# B&R Automation Studio project PT_KB_V01 (part 2)

#### Types.typ - Exported data types
```iecst
(* ============================================================================ *)
(* BR_LIB - CENTRALNI PREGLED SVIH DATA TYPE DEKLARACIJA                       *)
(* Sadrzi TYPE deklaracije iz FB-ova koje smo standardizovali.                  *)
(* Namena: referenca, copy/paste i priprema za eventualno centralno tipiziranje.*)
(* ============================================================================ *)

TYPE
	(* ======================================================================== *)
	(* FB_AI_01_DI_01                                                         *)
	(* ======================================================================== *)
	typInAI01_DI01 : STRUCT (* Ulazna struktura FB_AI_01_DI_01. *)
		Enable : BOOL; (* Globalni enable FB-a *)
		RawValue : INT; (* Raw vrednost sa AI kanala *)
		ManualValue : REAL; (* Rucno zadana skalirana vrednost *)
		EnableManual : BOOL; (* TRUE = koristi ManualValue umesto RawValue *)
		ResetAlarm : BOOL; (* Reset latched alarma *)
		ManualAlarm : BOOL; (* Spoljasnji/manual alarm signal *)
		UnderRange : BOOL; (* Sistemski signal: ulaz ispod opsega *)
		OverRange : BOOL; (* Sistemski signal: ulaz iznad opsega *)
		TransmitterStatus : BOOL; (* TRUE = transmiter ispravan; FALSE = fault sa transmitera *)
	END_STRUCT;

	typParAI01_DI01 : STRUCT (* Parametarska struktura FB_AI_01_DI_01. *)
		RawMin : INT; (* Donja granica raw opsega *)
		RawMax : INT; (* Gornja granica raw opsega *)
		ScaledMin : REAL; (* Donja granica skaliranog opsega *)
		ScaledMax : REAL; (* Gornja granica skaliranog opsega *)
		EnableStatusCheck : BOOL; (* TRUE = koristi TransmitterStatus u logici; FALSE = ignorise statusni DI signal *)
		UnitOfMeasure : STRING[80]; (* Jedinica mere za izlaznu vrednost *)
	END_STRUCT;

	typOutAI01_DI01 : STRUCT (* Izlazna struktura FB_AI_01_DI_01. *)
		ScaledValue : REAL; (* Skalirana inzenjerska vrednost *)
		Status : BOOL; (* TRUE = FB je omogucen, bez Stop-a, blokirajuceg fault-a i re-enable zahteva. *)
		State : USINT; (* Numericki kod stanja *)
		State_comment : STRING[80]; (* Trenutni opis stanja *)
		UnitOfMeasureOut : STRING[80]; (* Prosledjena jedinica mere *)
		TransmitterStatusIn : BOOL; (* Kopija ulaznog statusnog signala transmitera za HMI/SCADA *)
		FaultLatched : BOOL; (* Memorisan fault do validnog reset-a. *)
		FaultCondition : BOOL; (* Trenutni fault uslov u ovom scan-u. *)
		ResetAllowed : BOOL; (* TRUE kada fault moze biti resetovan bez ponovnog latche-ovanja. *)
		ConfigValid : BOOL; (* TRUE kada su opsezi validno konfigurirani. *)
		ConfigFaultText : STRING[80]; (* Opis prve nevalidne konfiguracije parametara. *)
		FaultCode : USINT; (* Kod memorisanog fault uzroka. *)
		FaultText : STRING[80]; (* Tekst memorisanog fault uzroka. *)
		Diag : STRING[80]; (* Kratak operativni tekst za HMI nadzor. *)
	END_STRUCT;

	typIntAI01_DI01 : STRUCT (* Interna radna struktura FB_AI_01_DI_01. *)
		FaultLatched : BOOL; (* Memorisan alarm dok se ne resetuje *)
		FaultCondition : BOOL; (* Trenutni fault uslov u ovom scan-u *)
		ActiveFaultCode : USINT; (* Trenutni aktivni fault kod u ovom scan-u. *)
		ScaleSpanRaw : REAL; (* Raspon raw opsega *)
		ScaleSpanScaled : REAL; (* Raspon skaliranog opsega *)
		ManualValueLimited : REAL; (* Ogranicena manual vrednost na parametarski opseg *)
		ResetRequest : BOOL; (* Interna kopija reset komande *)
		ResetAllowed : BOOL; (* Interna dozvola reset-a latched fault-a. *)
		ConfigValid : BOOL; (* FALSE kada opsezi nisu validno konfigurisani. *)
		ConfigFaultText : STRING[80]; (* Tekst prve nevalidne konfiguracije. *)
		FaultCode : USINT; (* Memorisani fault kod. *)
		FaultText : STRING[80]; (* Tekst memorisanog fault uzroka. *)
		Diag : STRING[80]; (* Interna dijagnostika trenutnog rezima i fault stanja. *)
	END_STRUCT;

	typConstAI01_DI01 : STRUCT (* Struktura konstanti i state tekstova FB_AI_01_DI_01. *)
		ST_DISABLED : USINT := 0; (* Blok onemogucen (Enable=FALSE). *)
		ST_ACTIVE : USINT := 1; (* Normalan rad bez alarma. *)
		ST_UNDERRANGE : USINT := 2; (* Raw vrednost ispod RawMin granice. *)
		ST_OVERRANGE : USINT := 3; (* Raw vrednost iznad RawMax granice. *)
		ST_FAULT : USINT := 4; (* Latched fault stanje u automatskom radu. *)
		ST_MANUAL : USINT := 5; (* Aktivno manuelno zadavanje bez fault-a. *)
		ST_MANUAL_FAULT : USINT := 6; (* Manuelni rad uz aktivan latched fault. *)
		ST_TRANSMITTER_STATUS_0 : USINT := 7; (* Statusni DI transmitera je FALSE. *)
		FLT_NONE : USINT := 0; (* Nema aktivnog fault uzroka. *)
		FLT_MANUAL_ALARM : USINT := 1; (* ManualAlarm ulaz je aktivan. *)
		FLT_UNDERRANGE : USINT := 2; (* UnderRange signal je aktivan. *)
		FLT_OVERRANGE : USINT := 3; (* OverRange signal je aktivan. *)
		FLT_CONFIG_INVALID : USINT := 4; (* Parametri opsega su nevalidni. *)
		CMT_DISABLED : STRING[80] := 'Stanje 0: transmiter neaktivan (Enable=FALSE), izlaz je na 0.0.'; (* Tekstualni opis stanja ST_DISABLED. *)
		CMT_ACTIVE : STRING[80] := 'Stanje 1: normalan rad, ulaz je u dozvoljenom opsegu, bez alarma.'; (* Tekstualni opis stanja ST_ACTIVE. *)
		CMT_UNDERRANGE : STRING[80] := 'Stanje 2: ulazna raw vrednost je ispod definisanog minimuma (RawMin).'; (* Tekstualni opis stanja ST_UNDERRANGE. *)
		CMT_OVERRANGE : STRING[80] := 'Stanje 3: ulazna raw vrednost je iznad definisanog maksimuma (RawMax).'; (* Tekstualni opis stanja ST_OVERRANGE. *)
		CMT_FAULT : STRING[80] := 'Stanje 4: prisutan je alarm (latched), potreban je ResetAlarm za potvrdu.'; (* Tekstualni opis stanja ST_FAULT. *)
		CMT_MANUAL : STRING[80] := 'Stanje 5: aktivan rucni rezim, ScaledValue dolazi iz ManualValue.'; (* Tekstualni opis stanja ST_MANUAL. *)
		CMT_MANUAL_FAULT : STRING[80] := 'Stanje 6: aktivan rucni rezim i istovremeno prisutan latched alarm.'; (* Tekstualni opis stanja ST_MANUAL_FAULT. *)
		CMT_TRANSMITTER_STATUS_0 : STRING[80] := 'Stanje 7: statusni DI signal transmitera je 0 (EnableStatusCheck=TRUE).'; (* Tekstualni opis stanja ST_TRANSMITTER_STATUS_0. *)
	END_STRUCT;

	typAI01_DI01 : STRUCT (* Agregatna struktura svih sekcija za FB_AI_01_DI_01. *)
		Input : typInAI01_DI01; (* Ulazni signali i komande bloka. *)
		Param : typParAI01_DI01; (* Parametri skaliranja i ponasanja. *)
		Output : typOutAI01_DI01; (* Izlazi, status i state informacije. *)
		Internal : typIntAI01_DI01; (* Interna radna memorija. *)
		Constant : typConstAI01_DI01; (* Konstante state kodova i tekstova. *)
	END_STRUCT;

	(* ======================================================================== *)
	(* FB_AI_01_DI_01_DO_02                                                    *)
	(* ======================================================================== *)
	typInAI01_DI01_DO02 : STRUCT (* Ulazna struktura FB_AI_01_DI_01_DO_02. *)
		Enable : BOOL; (* Globalni enable FB-a *)
		RawValue : INT; (* Raw vrednost sa AI kanala *)
		ManualValue : REAL; (* Rucno zadana skalirana vrednost *)
		EnableManual : BOOL; (* TRUE = koristi ManualValue umesto RawValue *)
		ResetAlarm : BOOL; (* Reset latched alarma *)
		ManualAlarm : BOOL; (* Spoljasnji/manual alarm signal *)
		UnderRange : BOOL; (* Sistemski signal: ulaz ispod opsega *)
		OverRange : BOOL; (* Sistemski signal: ulaz iznad opsega *)
		TransmitterStatus : BOOL; (* TRUE = transmiter ispravan; FALSE = fault sa transmitera *)
		RangeSelect : USINT; (* Izbor opsega 1..4 *)
		RangeSettleTime : TIME; (* Vreme stabilizacije nakon promene opsega *)
	END_STRUCT;

	typParAI01_DI01_DO02 : STRUCT (* Parametarska struktura FB_AI_01_DI_01_DO_02. *)
		RawMin : INT; (* Donja granica raw opsega *)
		RawMax : INT; (* Gornja granica raw opsega *)
		ScaledMin_R1 : REAL; (* Donja granica skaliranog opsega R1 *)
		ScaledMax_R1 : REAL; (* Gornja granica skaliranog opsega R1 *)
		ScaledMin_R2 : REAL; (* Donja granica skaliranog opsega R2 *)
		ScaledMax_R2 : REAL; (* Gornja granica skaliranog opsega R2 *)
		ScaledMin_R3 : REAL; (* Donja granica skaliranog opsega R3 *)
		ScaledMax_R3 : REAL; (* Gornja granica skaliranog opsega R3 *)
		ScaledMin_R4 : REAL; (* Donja granica skaliranog opsega R4 *)
		ScaledMax_R4 : REAL; (* Gornja granica skaliranog opsega R4 *)
		UnitOfMeasure : STRING[80]; (* Jedinica mere za izlaznu vrednost *)
	END_STRUCT;

	typOutAI01_DI01_DO02 : STRUCT (* Izlazna struktura FB_AI_01_DI_01_DO_02. *)
		ScaledValue : REAL; (* Skalirana inzenjerska vrednost *)
		Status : BOOL; (* TRUE = bez alarma i Enable=TRUE *)
		State : USINT; (* Numericki kod stanja *)
		State_comment : STRING[80]; (* Trenutni opis stanja *)
		UnitOfMeasureOut : STRING[80]; (* Prosledjena jedinica mere *)
		TransmitterStatusIn : BOOL; (* Kopija ulaznog statusnog signala transmitera za HMI/SCADA *)
		ActiveRange : USINT; (* Trenutno aktivan opseg 1..4 *)
		RangeComment : STRING[40]; (* Opis aktivnog opsega *)
		RangeBit0_out : BOOL; (* DO bit 0 za izbor opsega *)
		RangeBit1_out : BOOL; (* DO bit 1 za izbor opsega *)
		RangeChanging : BOOL; (* TRUE tokom stabilizacije promene opsega *)
		FaultProcessOut : BOOL; (* TRUE kada je aktivan procesni fault *)
		FaultConfigOut : BOOL; (* TRUE kada je aktivan konfiguracioni fault *)
	END_STRUCT;

	typIntAI01_DI01_DO02 : STRUCT (* Interna radna struktura FB_AI_01_DI_01_DO_02. *)
		FaultLatched : BOOL; (* Memorisan alarm dok se ne resetuje *)
		FaultCondition : BOOL; (* Trenutni fault uslov u ovom scan-u *)
		FaultProcess : BOOL; (* Procesni fault: DI status i under/over-range *)
		FaultConfig : BOOL; (* Konfiguracioni fault: parametri i range izbor *)
		ScaleSpanRaw : REAL; (* Raspon raw opsega *)
		ScaleSpanScaled : REAL; (* Raspon aktivnog skaliranog opsega *)
		ManualValueLimited : REAL; (* Ogranicena manual vrednost na aktivan opseg *)
		ActiveScaledMin : REAL; (* Donja granica aktivnog opsega *)
		ActiveScaledMax : REAL; (* Gornja granica aktivnog opsega *)
		LastGoodScaledValue : REAL; (* Poslednja validna vrednost pre promene opsega *)
		PrevRangeSelect : USINT; (* Prethodno izabrani opseg *)
		RangeChangeMem : BOOL; (* Memorija promene opsega *)
		ResetRequest : BOOL; (* Interna kopija reset komande *)
		RangeSettleTimeEffective : TIME; (* Validiran PT za tajmer stabilizacije *)
		RangeSettleTimer : TON; (* Tajmer stabilizacije posle promene opsega *)
	END_STRUCT;

	typConstAI01_DI01_DO02 : STRUCT (* Struktura konstanti i state tekstova FB_AI_01_DI_01_DO_02. *)
		ST_DISABLED : USINT := 0; (* Blok onemogucen (Enable=FALSE). *)
		ST_ACTIVE : USINT := 1; (* Normalan rad bez alarma. *)
		ST_UNDERRANGE : USINT := 2; (* Raw vrednost ispod RawMin granice. *)
		ST_OVERRANGE : USINT := 3; (* Raw vrednost iznad RawMax granice. *)
		ST_FAULT : USINT := 4; (* Latched fault stanje u automatskom radu. *)
		ST_MANUAL : USINT := 5; (* Aktivno manuelno zadavanje bez fault-a. *)
		ST_MANUAL_FAULT : USINT := 6; (* Manuelni rad uz aktivan latched fault. *)
		ST_TRANSMITTER_STATUS_0 : USINT := 7; (* Statusni DI transmitera je FALSE. *)
		ST_RANGE_CHANGING : USINT := 8; (* U toku je stabilizacija nakon promene opsega. *)
		CMT_DISABLED : STRING[80] := 'Stanje 0: transmiter neaktivan (Enable=FALSE), izlaz je na 0.0.'; (* Tekstualni opis stanja ST_DISABLED. *)
		CMT_ACTIVE : STRING[80] := 'Stanje 1: normalan rad, ulaz je u dozvoljenom opsegu, bez alarma.'; (* Tekstualni opis stanja ST_ACTIVE. *)
		CMT_UNDERRANGE : STRING[80] := 'Stanje 2: ulazna raw vrednost je ispod definisanog minimuma (RawMin).'; (* Tekstualni opis stanja ST_UNDERRANGE. *)
		CMT_OVERRANGE : STRING[80] := 'Stanje 3: ulazna raw vrednost je iznad definisanog maksimuma (RawMax).'; (* Tekstualni opis stanja ST_OVERRANGE. *)
		CMT_FAULT : STRING[80] := 'Stanje 4: prisutan je alarm (latched), potreban je ResetAlarm za potvrdu.'; (* Tekstualni opis stanja ST_FAULT. *)
		CMT_MANUAL : STRING[80] := 'Stanje 5: aktivan rucni rezim, ScaledValue dolazi iz ManualValue.'; (* Tekstualni opis stanja ST_MANUAL. *)
		CMT_MANUAL_FAULT : STRING[80] := 'Stanje 6: aktivan rucni rezim i istovremeno prisutan latched alarm.'; (* Tekstualni opis stanja ST_MANUAL_FAULT. *)
		CMT_TRANSMITTER_STATUS_0 : STRING[80] := 'Stanje 7: statusni DI signal transmitera je 0; skaliranje ostaje aktivno.'; (* Tekstualni opis stanja ST_TRANSMITTER_STATUS_0. *)
		CMT_RANGE_CHANGING : STRING[80] := 'Stanje 8: promena opsega je u toku; ceka se stabilizacija opsega.'; (* Tekstualni opis stanja ST_RANGE_CHANGING. *)
	END_STRUCT;

	typAI01_DI01_DO02 : STRUCT (* Agregatna struktura svih sekcija za FB_AI_01_DI_01_DO_02. *)
		Input : typInAI01_DI01_DO02; (* Ulazi sa izborom opsega i komandama. *)
		Param : typParAI01_DI01_DO02; (* Parametri opsega i skaliranja. *)
		Output : typOutAI01_DI01_DO02; (* Izlazi, aktivan opseg i fault status. *)
		Internal : typIntAI01_DI01_DO02; (* Interne pomocne promenljive i tajmeri. *)
		Constant : typConstAI01_DI01_DO02; (* Konstante stanja i komentari stanja. *)
	END_STRUCT;

	(* ======================================================================== *)
	(* FB_DI                                                                    *)
	(* ======================================================================== *)
	typInDI : STRUCT (* Ulazna struktura FB_DI. *)
		Enable : BOOL; (* Globalni enable FB-a *)
		SensorIn : BOOL; (* Digitalni ulaz sa terena *)
		StatusIn : BOOL; (* Statusni signal uredjaja, opciono koristi logika *)
		EnableManual : BOOL; (* TRUE = koristi ManualValue umesto SignalIn *)
		ManualValue : BOOL; (* Rucno zadat DI signal *)
		ResetAlarm : BOOL; (* Reset latched alarma *)
		ManualAlarm : BOOL; (* Spoljasnji/manual alarm signal *)
	END_STRUCT;

	typParDI : STRUCT (* Parametarska struktura FB_DI. *)
		UseStatusInput : BOOL; (* TRUE = proverava StatusIn; FALSE = ignorise ga *)
		InvertSignal : BOOL; (* TRUE = invertuje ulaznu DI vrednost *)
		DelayOn : TIME; (* Vreme potvrde OFF->ON prelaza *)
		DelayOff : TIME; (* Vreme potvrde ON->OFF prelaza *)
		AlarmOnTrue : BOOL; (* Alarm aktivan kada je Value=TRUE *)
		AlarmOnFalse : BOOL; (* Alarm aktivan kada je Value=FALSE *)
		TextTrue : STRING[80]; (* Tekst za stanje Value=TRUE *)
		TextFalse : STRING[80]; (* Tekst za stanje Value=FALSE *)
		TextAlarm : STRING[80]; (* Tekst za alarm stanje *)
		TextFault : STRING[80]; (* Tekst za fault stanje *)
	END_STRUCT;

	typOutDI : STRUCT (* Izlazna struktura FB_DI. *)
		Value : BOOL; (* Finalna DI vrednost nakon manual/invert/delay obrade *)
		Status : BOOL; (* TRUE = Enable aktivan i nema latched fault-a. *)
		Alarm : BOOL; (* Procesni alarm prema AlarmOnTrue/AlarmOnFalse *)
		Error : BOOL; (* Fault latch izlaz *)
		ManualActive : BOOL; (* TRUE kada je manual rezim aktivan *)
		State : USINT; (* Numericki kod stanja *)
		State_comment : STRING[80]; (* Tekstualni opis stanja *)
		StatusSignalIn : BOOL; (* Kopija statusnog signala za HMI/SCADA *)
		FaultLatched : BOOL; (* Memorisan fault do validnog reset-a *)
		FaultCondition : BOOL; (* Trenutni fault uslov u ovom scan-u *)
		AlarmCondition : BOOL; (* Trenutni procesni alarm uslov *)
		ResetAllowed : BOOL; (* TRUE kada fault moze biti resetovan bez ponovnog latche-ovanja. *)
		ConfigValid : BOOL; (* TRUE kada su DelayOn i DelayOff parametri validni. *)
		ConfigFaultText : STRING[80]; (* Opis nevalidne konfiguracije parametara. *)
		FaultCode : USINT; (* Kod memorisanog fault uzroka. *)
		FaultText : STRING[80]; (* Tekst memorisanog fault uzroka. *)
		Diag : STRING[80]; (* Kratak operativni tekst za HMI nadzor. *)
	END_STRUCT;

	typIntDI : STRUCT (* Interna radna struktura FB_DI. *)
		SignalRaw : BOOL; (* Vrednost pre delay obrade *)
		SignalFiltered : BOOL; (* Vrednost nakon delay obrade *)
		FaultLatched : BOOL; (* Interni fault latch *)
		FaultCondition : BOOL; (* Interni fault uslov u scan-u *)
		AlarmCondition : BOOL; (* Interni procesni alarm uslov *)
		ConfigValid : BOOL; (* FALSE kada su DelayOn/DelayOff parametri nevalidni. *)
		ResetAllowed : BOOL; (* Interna dozvola reseta fault-a. *)
		FaultCode : USINT; (* Memorisani kod fault uzroka. *)
		FaultText : STRING[80]; (* Tekst memorisanog fault uzroka. *)
		Diag : STRING[80]; (* Interna dijagnostika trenutnog rezima i fault stanja. *)
		TonOn : TON; (* Delay ON tajmer *)
		TonOff : TON; (* Delay OFF tajmer *)
	END_STRUCT;

	typConstDI : STRUCT (* Struktura state konstanti FB_DI. *)
		ST_DISABLED : USINT := 0; (* Blok onemogucen. *)
		ST_AUTO_FALSE : USINT := 1; (* Auto rezim, izlazna vrednost FALSE. *)
		ST_AUTO_TRUE : USINT := 2; (* Auto rezim, izlazna vrednost TRUE. *)
		ST_AUTO_ALARM : USINT := 3; (* Auto rezim sa procesnim alarmom. *)
		ST_AUTO_FAULT : USINT := 4; (* Auto rezim sa fault stanjem. *)
		ST_MAN_FALSE : USINT := 5; (* Manual rezim, izlazna vrednost FALSE. *)
		ST_MAN_TRUE : USINT := 6; (* Manual rezim, izlazna vrednost TRUE. *)
		ST_MAN_ALARM : USINT := 7; (* Manual rezim sa procesnim alarmom. *)
		ST_MAN_FAULT : USINT := 8; (* Manual rezim sa fault stanjem. *)
		FLT_NONE : USINT := 0; (* Nema aktivnog fault uzroka. *)
		FLT_MANUAL_ALARM : USINT := 1; (* ManualAlarm ulaz je aktivan. *)
		FLT_STATUS_INPUT : USINT := 2; (* StatusIn fault kada je UseStatusInput aktivan. *)
		FLT_CONFIG_INVALID : USINT := 3; (* Delay parametri su nevalidni. *)
	END_STRUCT;

	typDI : STRUCT (* Agregatna struktura svih sekcija za FB_DI. *)
		Input : typInDI; (* Ulazni signali, manual i reset komande. *)
		Param : typParDI; (* Parametri obrade i tekstovi stanja. *)
		Output : typOutDI; (* Finalna DI vrednost, alarm/fault i stanje. *)
		Internal : typIntDI; (* Interna logika filtracije i latch-a. *)
		Constant : typConstDI; (* Konstante state kodova DI bloka. *)
	END_STRUCT;

	(* ======================================================================== *)
	(* FB_V_ON_OFF_FB                                                           *)
	(* ======================================================================== *)
	typInVOnOff : STRUCT (* Ulazna struktura FB_V_ON_OFF_FB. *)
		Enable : BOOL; (* Globalni enable FB-a *)
		Stop : BOOL; (* Operativni stop: odmah deaktivira kalem i zahteva novi Enable ciklus. *)
		EnableManual : BOOL; (* TRUE = komanda pozicije dolazi iz manual ulaza *)
		Open_Manual : BOOL; (* Manual zahtev: TRUE otvori, FALSE zatvori *)
		OpenFb : BOOL; (* Povratni signal otvorenog krajnjeg polozaja *)
		CloseFb : BOOL; (* Povratni signal zatvorenog krajnjeg polozaja *)
		ResetAlarm : BOOL; (* Reset memorisanog alarma, samo kada trenutni fault uslov nije aktivan *)
		ManualAlarm : BOOL; (* Spoljni/manual fault zahtev *)
		ForceCmd : BOOL; (* TRUE = komanda prolazi ka ventilu i u fault stanju; FALSE = komanda blokirana (bezbedan polozaj) *)
	END_STRUCT;

	typParVOnOff : STRUCT (* Parametarska struktura FB_V_ON_OFF_FB. *)
		DeEnergizedOpen : BOOL; (* TRUE = ventil je bez napajanja otvoren; FALSE = bez napajanja zatvoren. *)
		FbOpenExists : BOOL; (* TRUE ako fizicki postoji Open feedback signal *)
		FbCloseExists : BOOL; (* TRUE ako fizicki postoji Close feedback signal *)
		OpenMinTime : TIME; (* Minimalno dozvoljeno vreme otvaranja pre OpenFb potvrde *)
		OpenMaxTime : TIME; (* Maksimalno dozvoljeno vreme otvaranja do OpenFb potvrde *)
		CloseMinTime : TIME; (* Minimalno dozvoljeno vreme zatvaranja pre CloseFb potvrde *)
		CloseMaxTime : TIME; (* Maksimalno dozvoljeno vreme zatvaranja do CloseFb potvrde *)
		StableFbDelay : TIME; (* Delay za detekciju nestabilnog feedback-a u stabilnim stanjima *)
	END_STRUCT;

	typOutVOnOff : STRUCT (* Izlazna struktura FB_V_ON_OFF_FB. *)
		Cmd : BOOL; (* Komanda jednom kalemu; funkcija zavisi od DeEnergizedOpen. *)
		Opened : BOOL; (* FB trenutno koristi otvoren polozaj, fizicki potvrdjen ili vremenski pretpostavljen. *)
		Closed : BOOL; (* FB trenutno koristi zatvoren polozaj, fizicki potvrdjen ili vremenski pretpostavljen. *)
		PositionConfirmed : BOOL; (* Aktivni krajnji polozaj je potvrdjen odgovarajucim fizickim feedback-om. *)
		PositionAssumed : BOOL; (* Aktivni krajnji polozaj je vremenski pretpostavljen bez odgovarajuceg feedback-a. *)
		OpenAssumed : BOOL; (* Otvoren polozaj je vremenski pretpostavljen. *)
		CloseAssumed : BOOL; (* Zatvoren polozaj je vremenski pretpostavljen. *)
		Status : BOOL; (* TRUE = bez alarma i Enable=TRUE *)
		InTransition : BOOL; (* TRUE dok je ventil u stanjima ST_OPENING ili ST_CLOSING *)
		StopActive : BOOL; (* Kopija aktivnog operativnog Stop zahteva. *)
		WaitingReEnable : BOOL; (* FB ceka novi Enable FALSE->TRUE ciklus posle Stop-a ili fault reseta. *)
		ResetAllowed : BOOL; (* TRUE kada je dozvoljen reset latched alarma *)
		State : USINT; (* Kopija internog stanja za HMI *)
		State_comment : STRING[80]; (* Opis stanja za HMI *)
		Diag : STRING[40]; (* Kratka operativna dijagnostika za live nadzor *)
		FaultLatched : BOOL; (* Memorisan alarm, ostaje 1 do validnog reseta *)
		FaultCondition : BOOL; (* Trenutni fault uslov u ovom scan-u *)
		FaultInManual : BOOL; (* Alarm je nastao dok je bio aktivan manual mod *)
		FaultCode : USINT; (* Numericki kod alarma *)
		FaultText : STRING[80]; (* Tekst alarma za HMI *)
		ForceActive : BOOL; (* TRUE = blokirajuci fault je aktivan, a ForceCmd dozvoljava komandu. *)
		FeedbackAlarmCondition : BOOL; (* Trenutno nedostaje ocekivani stabilni feedback. *)
		FeedbackAlarmLatched : BOOL; (* Memorisan neblokirajuci alarm stabilnog feedback-a. *)
		FeedbackAlarmCode : USINT; (* Numericki kod neblokirajuceg feedback alarma. *)
		FeedbackAlarmText : STRING[80]; (* Tekst neblokirajuceg feedback alarma. *)
		ConfigFaultText : STRING[80]; (* Opis prve nevalidne konfiguracione vrednosti. *)
		LastOpenStartTime  : REAL; (* Vreme od Open komande do gubitka CloseFb [s]; 0.0 ako FbCloseExists=FALSE *)
		LastOpenTime       : REAL; (* Vreme od Open komande do OpenConfirm=TRUE [s]; 0.0 ako FbOpenExists=FALSE *)
		LastCloseStartTime : REAL; (* Vreme od ukidanja Open komande do gubitka OpenFb [s]; 0.0 ako FbOpenExists=FALSE *)
		LastCloseTime      : REAL; (* Vreme od ukidanja Open komande do CloseConfirm=TRUE [s]; 0.0 ako FbCloseExists=FALSE *)
	END_STRUCT;

	typIntVOnOff : STRUCT (* Interna radna struktura FB_V_ON_OFF_FB. *)
		DesiredOpen : BOOL; (* Zeljen polozaj ventila: TRUE = otvoren, FALSE = zatvoren *)
		CmdRequest : BOOL; (* Zahtev aktiviranja kalema nakon NC/NO konverzije. *)
		FaultLatched : BOOL; (* Memorisan alarm - ostaje aktivan dok se ne resetuje *)
		FaultCondition : BOOL; (* Trenutno aktivan uslov alarma u ovom ciklusu *)
		FaultInManual : BOOL; (* Pamti da li je alarm nastao u rucnom modu *)
		FaultCode : USINT; (* Interni broj greske *)
		FaultText : STRING[80]; (* Tekstualni opis greske za HMI *)
		OpenConfirm : BOOL; (* Potvrda da je ventil otvoren *)
		CloseConfirm : BOOL; (* Potvrda da je ventil zatvoren *)
		OpenAssumed : BOOL; (* Memorija vremenski pretpostavljenog otvorenog polozaja. *)
		CloseAssumed : BOOL; (* Memorija vremenski pretpostavljenog zatvorenog polozaja. *)
		FeedbackAlarmCondition : BOOL; (* Trenutni uslov neblokirajuceg feedback alarma. *)
		FeedbackAlarmLatched : BOOL; (* Memorisan neblokirajuci feedback alarm. *)
		FeedbackAlarmCode : USINT; (* Kod neblokirajuceg feedback alarma. *)
		ReEnableRequired : BOOL; (* Posle Stop-a ili fault reseta zahteva novi Enable rising edge. *)
		Step : USINT; (* Interno stanje state machine *)
		PrevEnable : BOOL; (* Pamti prethodno stanje Enable signala zbog detekcije rising edge *)
		OpeningStarted : BOOL; (* Tokom otvaranja: ventil je poceo da se otvara *)
		ClosingStarted : BOOL; (* Tokom zatvaranja: ventil je poceo da se zatvara *)
		StableClosedFbError : BOOL; (* U stabilno zatvorenom stanju postoji greska feedback-a *)
		StableOpenedFbError : BOOL; (* U stabilno otvorenom stanju postoji greska feedback-a *)
		OpenMinTimer : TON; (* Minimalno dozvoljeno vreme otvaranja *)
		OpenMaxTimer : TON; (* Maksimalno dozvoljeno vreme otvaranja *)
		CloseMinTimer : TON; (* Minimalno dozvoljeno vreme zatvaranja *)
		CloseMaxTimer : TON; (* Maksimalno dozvoljeno vreme zatvaranja *)
		OpenMeasureTimer : TON; (* Merenje realnog trajanja otvaranja *)
		CloseMeasureTimer : TON; (* Merenje realnog trajanja zatvaranja *)
		StableClosedFbTimer : TON; (* Delay za potvrdu greske feedback-a u zatvorenom stanju *)
		StableOpenedFbTimer : TON; (* Delay za potvrdu greske feedback-a u otvorenom stanju *)
		PrevCloseFb : BOOL; (* Prethodni scan CloseFb - za detekciju falling edge u ST_OPENING *)
		PrevOpenFb  : BOOL; (* Prethodni scan OpenFb  - za detekciju falling edge u ST_CLOSING *)
	END_STRUCT;

	typCfgVOnOff : STRUCT (* Konfiguraciona struktura state/fault kodova FB_V_ON_OFF_FB. *)
		OpenMinTime_Valid : TIME; (* Validirano minimalno vreme otvaranja. *)
		OpenMaxTime_Valid : TIME; (* Validirano maksimalno vreme otvaranja. *)
		CloseMinTime_Valid : TIME; (* Validirano minimalno vreme zatvaranja. *)
		CloseMaxTime_Valid : TIME; (* Validirano maksimalno vreme zatvaranja. *)
		StableFbDelay_Valid : TIME; (* Validiran delay nadzora stabilnog feedback-a. *)

		ST_DISABLED : USINT := 0; (* Blok onemogucen. *)
		ST_IDLE_CLOSED : USINT := 10; (* Stabilno stanje: ventil zatvoren. *)
		ST_IDLE_OPENED : USINT := 20; (* Stabilno stanje: ventil otvoren. *)
		ST_OPENING : USINT := 30; (* Tranzicija otvaranja u toku. *)
		ST_CLOSING : USINT := 40; (* Tranzicija zatvaranja u toku. *)
		ST_STOPPED : USINT := 50; (* Operativni Stop je aktivan. *)
		ST_WAIT_REENABLE : USINT := 60; (* Ceka se novi Enable FALSE->TRUE ciklus. *)
		ST_FAULT : USINT := 90; (* Fault stanje ventila. *)

		FLT_NONE : USINT := 0; (* Nema aktivnog fault-a. *)
		FLT_MANUAL_ALARM : USINT := 1; (* Manual alarm zahtev je aktivan. *)
		FLT_FB_CONFLICT : USINT := 2; (* Konflikt feedback-a (OpenFb i CloseFb). *)
		FLT_OPEN_TIMEOUT : USINT := 3; (* Otvaranje nije potvrdjeno u OpenMaxTime. *)
		FLT_OPEN_TOO_FAST : USINT := 4; (* Otvaranje potvrdeno pre OpenMinTime. *)
		FLT_CLOSE_TIMEOUT : USINT := 5; (* Zatvaranje nije potvrdjeno u CloseMaxTime. *)
		FLT_CLOSE_TOO_FAST : USINT := 6; (* Zatvaranje potvrdeno pre CloseMinTime. *)
		FLT_TIME_CONFIG_INVALID : USINT := 9; (* Nevalidna konfiguracija vremenskih parametara. *)

		FB_ALM_NONE : USINT := 0; (* Nema neblokirajuceg feedback alarma. *)
		FB_ALM_STABLE_OPEN_LOST : USINT := 1; (* Izgubljen OpenFb u stabilno otvorenom stanju. *)
		FB_ALM_STABLE_CLOSE_LOST : USINT := 2; (* Izgubljen CloseFb u stabilno zatvorenom stanju. *)
	END_STRUCT;

	(* ======================================================================== *)
	(* FB_V_EMV (elektromotorni ventil sa odvojenim OPEN/CLOSE komandama)       *)
	(* ======================================================================== *)
	typInVEmv : STRUCT (* Ulazna struktura FB_V_EMV. *)
		Enable : BOOL; (* Globalna dozvola rada FB-a. *)
		Stop : BOOL; (* Operativni stop: odmah gasi obe komande bez generisanja fault-a. *)
		EnableManual : BOOL; (* TRUE = koristi OpenManual umesto automatskog Open zahteva. *)
		OpenManual : BOOL; (* Manualni zahtev polozaja: TRUE = OPEN, FALSE = CLOSE. *)
		ForceCmd : BOOL; (* Dozvola kontrolisanog kretanja u suprotnom smeru iz fault-a. *)
		ResetAlarm : BOOL; (* Zahtev za reset latched fault-a kada su ispunjeni bezbedni uslovi. *)
		ManualAlarm : BOOL; (* Spoljasnji fault/interlock zahtev. *)
		LampOpen : BOOL; (* Fabricki OPEN kraj hoda, klema 9; postoji samo uz OPEN komandni lanac. *)
		LampClose : BOOL; (* Fabricki CLOSE kraj hoda, klema 8; postoji samo uz CLOSE komandni lanac. *)
		OpenFb : BOOL; (* Trajna pomocna potvrda otvorenog polozaja AOLS. *)
		CloseFb : BOOL; (* Trajna pomocna potvrda zatvorenog polozaja ACLS. *)
		OverTorque : BOOL; (* Opcioni signal prekomernog momenta aktuatora. *)
	END_STRUCT;

	typParVEmv : STRUCT (* Parametarska struktura FB_V_EMV. *)
		LampOpenExists : BOOL; (* TRUE ako je signal fabriskog OPEN kraja hoda dostupan PLC-u. *)
		LampCloseExists : BOOL; (* TRUE ako je signal fabriskog CLOSE kraja hoda dostupan PLC-u. *)
		OpenFbExists : BOOL; (* TRUE ako postoji trajni OpenFb/AOLS signal. *)
		CloseFbExists : BOOL; (* TRUE ako postoji trajni CloseFb/ACLS signal. *)
		OverTorqueExists : BOOL; (* TRUE ako je OverTorque signal fizicki dostupan i proveren. *)
		UnexpectedOpenLimitCheck : BOOL; (* TRUE = neocekivani LampOpen tokom zatvaranja generise fault. *)
		UnexpectedCloseLimitCheck : BOOL; (* TRUE = neocekivani LampClose tokom otvaranja generise fault. *)
		OpenMaxTime : TIME; (* Maksimalno vreme otvaranja ili vremenski hod kada nema OPEN signala. *)
		CloseMaxTime : TIME; (* Maksimalno vreme zatvaranja ili vremenski hod kada nema CLOSE signala. *)
		DeadTime : TIME; (* Obavezno vreme sa obe komande na FALSE pre promene/pokretanja smera. *)
		EndLimitFilterTime : TIME; (* Stabilizacioni filter za LampOpen i LampClose. *)
		PositionFbFilterTime : TIME; (* Stabilizacioni filter za OpenFb i CloseFb. *)
		OverTorqueFilterTime : TIME; (* Stabilizacioni filter OverTorque signala; T#0ms je dozvoljeno. *)
		PositionConfirmTime : TIME; (* Vreme cekanja trajnog Fb nakon fabriskog kraja hoda. *)
		StableFbLossTime : TIME; (* Dozvoljeno vreme gubitka potvrde u idle stanju; T#0ms je dozvoljeno. *)
	END_STRUCT;

	typOutVEmv : STRUCT (* Izlazna struktura FB_V_EMV. *)
		CmdOpen : BOOL; (* Komanda PLC izlazu za otvaranje. *)
		CmdClose : BOOL; (* Komanda PLC izlazu za zatvaranje. *)
		Opened : BOOL; (* TRUE samo za fizicki potvrdjen otvoren polozaj. *)
		Closed : BOOL; (* TRUE samo za fizicki potvrdjen zatvoren polozaj. *)
		OpenAssumed : BOOL; (* Otvoren polozaj je vremenski pretpostavljen bez OpenFb. *)
		CloseAssumed : BOOL; (* Zatvoren polozaj je vremenski pretpostavljen bez CloseFb. *)
		Intermediate : BOOL; (* Ventil nije potvrdjeno ni otvoren ni zatvoren. *)
		Position : USINT; (* Numericki kod polozaja. *)
		PositionText : STRING[80]; (* Tekstualni opis numerickog koda polozaja. *)
		PositionConfirmed : BOOL; (* Trenutni krajnji polozaj je fizicki potvrdjen. *)
		PositionAssumed : BOOL; (* Trenutni krajnji polozaj je samo vremenski pretpostavljen. *)
		Status : BOOL; (* FB je omogucen i nema latched fault-a. *)
		Ready : BOOL; (* FB je sinhronizovan i spreman za regularnu komandu. *)
		InTransition : BOOL; (* Aktivna je regularna ili force sekvenca kretanja. *)
		Opening : BOOL; (* Aktivna je sekvenca otvaranja. *)
		Closing : BOOL; (* Aktivna je sekvenca zatvaranja. *)
		Stopped : BOOL; (* FB se nalazi u ST_STOPPED. *)
		StopActive : BOOL; (* Kopija aktivnog operativnog Stop zahteva. *)
		InitActive : BOOL; (* Aktivna je pocetna sinhronizacija polozaja. *)
		WaitingReEnable : BOOL; (* FB ceka novi Enable FALSE->TRUE ciklus. *)
		DeadTimeActive : BOOL; (* Aktivna je obavezna pauza sa obe komande ugasene. *)
		WaitingPositionConfirm : BOOL; (* Ceka se trajni feedback nakon fabriskog kraja hoda. *)
		ManualActive : BOOL; (* Aktivno je manualno zadavanje. *)
		ForceAllowed : BOOL; (* Uslovi dozvoljavaju force kretanje u suprotnom smeru. *)
		ForceActive : BOOL; (* Force kretanje ili force dead-time je aktivan. *)
		ForceBlocked : BOOL; (* Force zahtev postoji, ali ga zastitni uslovi blokiraju. *)
		DesiredOpen : BOOL; (* Finalni zahtev nakon auto/manual izbora. *)
		State : USINT; (* Numericki kod aktivnog stanja. *)
		State_comment : STRING[80]; (* Tekstualni opis numerickog state koda. *)
		Diag : STRING[80]; (* Kratak operativni opis trenutnog dogadjaja. *)
		FaultCondition : BOOL; (* Trenutni fault uslov postoji u ovom scan-u. *)
		FaultLatched : BOOL; (* Fault je memorisan do validnog reseta. *)
		ResetAllowed : BOOL; (* Trenutno su ispunjeni uslovi za reset. *)
		FaultCode : USINT; (* Numericki kod originalnog latched fault-a. *)
		FaultText : STRING[80]; (* Tekstualni opis originalnog fault koda. *)
		FaultDirection : USINT; (* Smer u kojem je originalni fault nastao. *)
		FaultDirectionText : STRING[30]; (* Tekstualni opis smera originalnog fault-a. *)
		FaultInManual : BOOL; (* Fault je nastao u manualnom rezimu. *)
		FaultInForce : BOOL; (* Fault je nastao tokom force oporavka. *)
		ForceDirection : USINT; (* Dozvoljeni/aktivni smer force oporavka. *)
		ForceDirectionText : STRING[30]; (* Tekstualni opis force smera. *)
		ForceDiag : STRING[80]; (* Razlog dozvoljenog ili blokiranog force kretanja. *)
		RecoveryFaultCode : USINT; (* Kod novog fault-a nastalog tokom force oporavka. *)
		RecoveryFaultText : STRING[80]; (* Tekst novog fault-a tokom force oporavka. *)
		ConfigFaultText : STRING[80]; (* Precizan opis nevalidnog konfiguracionog parametra. *)
		OpenEndReached : BOOL; (* Memorija fabriskog OPEN kraja u aktuelnoj sekvenci. *)
		CloseEndReached : BOOL; (* Memorija fabriskog CLOSE kraja u aktuelnoj sekvenci. *)
		OpenFbStable : BOOL; (* Filtrirana stabilna vrednost OpenFb. *)
		CloseFbStable : BOOL; (* Filtrirana stabilna vrednost CloseFb. *)
		OverTorqueActive : BOOL; (* Filtriran i konfiguraciono omogucen OverTorque. *)
		CurrentTravelTime : REAL; (* Trenutno vreme aktivnog hoda [s]. *)
		LastOpenStartTime : REAL; (* Vreme od CmdOpen do gubitka CloseFb [s]. *)
		LastOpenTime : REAL; (* Vreme od CmdOpen do konfigurisanog OPEN kraja [s]. *)
		LastOpenFbTime : REAL; (* Vreme od CmdOpen do stabilnog OpenFb [s]. *)
		LastCloseStartTime : REAL; (* Vreme od CmdClose do gubitka OpenFb [s]. *)
		LastCloseTime : REAL; (* Vreme od CmdClose do konfigurisanog CLOSE kraja [s]. *)
		LastCloseFbTime : REAL; (* Vreme od CmdClose do stabilnog CloseFb [s]. *)
		LastOpenFbOffset : REAL; (* SIGNED [s]: OpenFb vreme minus LampOpen vreme; negativno = Fb je stigao ranije. *)
		OpenFbOffsetValid : BOOL; (* TRUE kada su oba OPEN dogadjaja izmerena u istom hodu. *)
		LastCloseFbOffset : REAL; (* SIGNED [s]: CloseFb vreme minus LampClose vreme; negativno = Fb je stigao ranije. *)
		CloseFbOffsetValid : BOOL; (* TRUE kada su oba CLOSE dogadjaja izmerena u istom hodu. *)
	END_STRUCT;

	typIntVEmv : STRUCT (* Interna radna struktura FB_V_EMV. *)
		DesiredOpen : BOOL; (* Finalni auto/manual zahtev polozaja. *)
		Step : USINT; (* Aktivno stanje state machine. *)
		NextDirection : USINT; (* Smer koji sledi nakon dead-time-a. *)
		PrevDirection : USINT; (* Poslednji aktivni smer motora. *)
		PrevEnable : BOOL; (* Prethodno stanje Enable signala. *)
		FaultCondition : BOOL; (* Trenutni fault uslov. *)
		FaultLatched : BOOL; (* Memorisan originalni fault. *)
		FaultCode : USINT; (* Kod originalnog fault-a. *)
		FaultDirection : USINT; (* Smer originalnog fault-a. *)
		FaultInManual : BOOL; (* Originalni fault je nastao u manualnom rezimu. *)
		FaultInForce : BOOL; (* Novi fault je nastao tokom force oporavka. *)
		RecoveryFaultCode : USINT; (* Novi fault tokom force oporavka. *)
		ConfigValid : BOOL; (* Svi parametri su validni. *)
		ConfigFaultText : STRING[80]; (* Opis prve detektovane konfiguracione greske. *)
		LampOpenStable : BOOL; (* Filtriran LampOpen signal. *)
		LampCloseStable : BOOL; (* Filtriran LampClose signal. *)
		OpenFbStable : BOOL; (* Filtriran OpenFb signal. *)
		CloseFbStable : BOOL; (* Filtriran CloseFb signal. *)
		OverTorqueStable : BOOL; (* Filtriran OverTorque signal. *)
		PrevOpenFbStable : BOOL; (* Prethodna filtrirana vrednost OpenFb. *)
		PrevCloseFbStable : BOOL; (* Prethodna filtrirana vrednost CloseFb. *)
		PrevOpenFbRaw : BOOL; (* Prethodna sirova vrednost OpenFb za merenje ivice. *)
		PrevCloseFbRaw : BOOL; (* Prethodna sirova vrednost CloseFb za merenje ivice. *)
		PrevLampOpenRaw : BOOL; (* Prethodna sirova vrednost LampOpen za merenje ivice. *)
		PrevLampCloseRaw : BOOL; (* Prethodna sirova vrednost LampClose za merenje ivice. *)
		OpenEndReached : BOOL; (* Memorija LampOpen dogadjaja u aktuelnom hodu. *)
		CloseEndReached : BOOL; (* Memorija LampClose dogadjaja u aktuelnom hodu. *)
		OpenFbSeen : BOOL; (* OpenFb je registrovan u aktuelnom OPEN hodu. *)
		CloseFbSeen : BOOL; (* CloseFb je registrovan u aktuelnom CLOSE hodu. *)
		OpenLampSeen : BOOL; (* LampOpen je registrovan u aktuelnom OPEN hodu. *)
		CloseLampSeen : BOOL; (* LampClose je registrovan u aktuelnom CLOSE hodu. *)
		OpenStartMeasured : BOOL; (* Gubitak CloseFb je izmeren u aktuelnom OPEN hodu. *)
		CloseStartMeasured : BOOL; (* Gubitak OpenFb je izmeren u aktuelnom CLOSE hodu. *)
		OpenFbEventTime : REAL; (* Vreme pojave OpenFb u aktuelnom hodu [s]. *)
		CloseFbEventTime : REAL; (* Vreme pojave CloseFb u aktuelnom hodu [s]. *)
		OpenLampEventTime : REAL; (* Vreme pojave LampOpen u aktuelnom hodu [s]. *)
		CloseLampEventTime : REAL; (* Vreme pojave LampClose u aktuelnom hodu [s]. *)
		ForceAllowed : BOOL; (* Izracunata dozvola force kretanja. *)
		ForceDirection : USINT; (* Izracunati suprotni smer force oporavka. *)
		ForceRequested : BOOL; (* ForceCmd i zahtev su uskladjeni sa suprotnim smerom. *)
		ForceRecoveryDone : BOOL; (* Uspesan force oporavak zavrsen; ceka se otpustanje ForceCmd. *)
		LampOpenFilterTimer : TON; (* Filter LampOpen signala. *)
		LampCloseFilterTimer : TON; (* Filter LampClose signala. *)
		OpenFbFilterTimer : TON; (* Filter OpenFb signala. *)
		CloseFbFilterTimer : TON; (* Filter CloseFb signala. *)
		OverTorqueFilterTimer : TON; (* Filter OverTorque signala. *)
		InitSyncTimer : TON; (* Cekanje stabilizacije ulaza u ST_INIT_SYNC. *)
		DeadTimeTimer : TON; (* Obavezna pauza izmedju smerova. *)
		OpenTravelTimer : TON; (* Nadzor maksimalnog vremena otvaranja. *)
		CloseTravelTimer : TON; (* Nadzor maksimalnog vremena zatvaranja. *)
		OpenConfirmTimer : TON; (* Cekanje OpenFb nakon LampOpen. *)
		CloseConfirmTimer : TON; (* Cekanje CloseFb nakon LampClose. *)
		StableOpenLossTimer : TON; (* Nadzor gubitka OpenFb u otvorenom idle stanju. *)
		StableCloseLossTimer : TON; (* Nadzor gubitka CloseFb u zatvorenom idle stanju. *)
	END_STRUCT;

	typCfgVEmv : STRUCT (* Konfiguraciona struktura FB_V_EMV. *)
		OpenMaxTimeValid : TIME; (* Validirano maksimalno vreme otvaranja. *)
		CloseMaxTimeValid : TIME; (* Validirano maksimalno vreme zatvaranja. *)
		DeadTimeValid : TIME; (* Validirano mrtvo vreme, najmanje T#500ms. *)
		EndLimitFilterTimeValid : TIME; (* Validirano vreme filtera fabriskih krajeva. *)
		PositionFbFilterTimeValid : TIME; (* Validirano vreme filtera trajnih potvrda. *)
		OverTorqueFilterTimeValid : TIME; (* Validirano vreme filtera momenta. *)
		PositionConfirmTimeValid : TIME; (* Validirano vreme cekanja trajne potvrde. *)
		StableFbLossTimeValid : TIME; (* Validirano vreme gubitka stabilne potvrde. *)
		ST_DISABLED : USINT := 0; (* FB nije omogucen. *)
		ST_INIT_SYNC : USINT := 5; (* Pocetna sinhronizacija bez komandovanja. *)
		ST_IDLE_CLOSED : USINT := 10; (* Fizicki potvrdjen zatvoren polozaj. *)
		ST_IDLE_OPENED : USINT := 20; (* Fizicki potvrdjen otvoren polozaj. *)
		ST_IDLE_CLOSE_ASSUMED : USINT := 30; (* Vremenski pretpostavljen zatvoren polozaj. *)
		ST_IDLE_OPEN_ASSUMED : USINT := 40; (* Vremenski pretpostavljen otvoren polozaj. *)
		ST_INTERMEDIATE : USINT := 50; (* Nepoznat ili medjupolozaj. *)
		ST_DIRECTION_DEADTIME : USINT := 60; (* Pauza pre regularnog smera. *)
		ST_OPENING : USINT := 70; (* Regularno otvaranje. *)
		ST_CLOSING : USINT := 80; (* Regularno zatvaranje. *)
		ST_WAIT_OPEN_CONFIRM : USINT := 90; (* Cekanje OpenFb nakon LampOpen. *)
		ST_WAIT_CLOSE_CONFIRM : USINT := 100; (* Cekanje CloseFb nakon LampClose. *)
		ST_STOPPED : USINT := 110; (* Operativni Stop je aktivan. *)
		ST_WAIT_REENABLE : USINT := 120; (* Cekanje novog Enable ciklusa. *)
		ST_FAULT : USINT := 200; (* Latched fault, obe komande ugasene. *)
		ST_FORCE_DEADTIME : USINT := 210; (* Pauza pre force oporavka. *)
		ST_FORCE_OPENING : USINT := 220; (* Force otvaranje iz CLOSE fault-a. *)
		ST_FORCE_CLOSING : USINT := 230; (* Force zatvaranje iz OPEN fault-a. *)
		ST_FORCE_WAIT_OPEN_CONFIRM : USINT := 240; (* Force OPEN zavrsen, ceka se OpenFb. *)
		ST_FORCE_WAIT_CLOSE_CONFIRM : USINT := 250; (* Force CLOSE zavrsen, ceka se CloseFb. *)
		POS_UNKNOWN : USINT := 0; (* Polozaj nije poznat. *)
		POS_CLOSED_CONFIRMED : USINT := 1; (* Zatvoren polozaj fizicki potvrdjen. *)
		POS_OPENED_CONFIRMED : USINT := 2; (* Otvoren polozaj fizicki potvrdjen. *)
		POS_INTERMEDIATE : USINT := 3; (* Ventil je u medjupolozaju. *)
		POS_CLOSED_ASSUMED : USINT := 4; (* Zatvoren polozaj vremenski pretpostavljen. *)
		POS_OPENED_ASSUMED : USINT := 5; (* Otvoren polozaj vremenski pretpostavljen. *)
		POS_CONFLICT : USINT := 6; (* OpenFb i CloseFb su istovremeno aktivni. *)
		DIR_NONE : USINT := 0; (* Nema aktivnog/poznatog smera. *)
		DIR_OPEN : USINT := 1; (* Smer otvaranja. *)
		DIR_CLOSE : USINT := 2; (* Smer zatvaranja. *)
		FLT_NONE : USINT := 0; (* Nema fault-a. *)
		FLT_MANUAL_ALARM : USINT := 1; (* Spoljasnji ManualAlarm je aktivan. *)
		FLT_OVER_TORQUE : USINT := 2; (* Aktivirana momentna zastita. *)
		FLT_POSITION_CONFLICT : USINT := 3; (* OpenFb i CloseFb su istovremeno aktivni. *)
		FLT_OUTPUT_CONFLICT : USINT := 4; (* CmdOpen i CmdClose su istovremeno izracunati. *)
		FLT_OPEN_TIMEOUT : USINT := 5; (* Nije dostignut OPEN kraj u OpenMaxTime. *)
		FLT_CLOSE_TIMEOUT : USINT := 6; (* Nije dostignut CLOSE kraj u CloseMaxTime. *)
		FLT_OPEN_CONFIRM_TIMEOUT : USINT := 7; (* LampOpen dostignut, ali OpenFb nije potvrdjen. *)
		FLT_CLOSE_CONFIRM_TIMEOUT : USINT := 8; (* LampClose dostignut, ali CloseFb nije potvrdjen. *)
		FLT_OPEN_FB_LOST : USINT := 9; (* OpenFb izgubljen u stabilno otvorenom stanju. *)
		FLT_CLOSE_FB_LOST : USINT := 10; (* CloseFb izgubljen u stabilno zatvorenom stanju. *)
		FLT_INVALID_CONFIG : USINT := 11; (* Parametri FB-a nisu validni. *)
		FLT_UNEXPECTED_OPEN_LIMIT : USINT := 12; (* LampOpen aktivan tokom zatvaranja. *)
		FLT_UNEXPECTED_CLOSE_LIMIT : USINT := 13; (* LampClose aktivan tokom otvaranja. *)
	END_STRUCT;

	typVEmv : STRUCT (* Agregatna struktura svih sekcija FB_V_EMV. *)
		Input : typInVEmv; (* Ulazni signali, rezimi i zastite. *)
		Param : typParVEmv; (* Parametri konfiguracije i vremena. *)
		Output : typOutVEmv; (* Komande, status, dijagnostika i merenja. *)
		Internal : typIntVEmv; (* Interna state machine memorija i tajmeri. *)
		Cfg : typCfgVEmv; (* Konstante stanja, polozaja, smerova i fault-ova. *)
	END_STRUCT;

	(* ======================================================================== *)
	(* FB_HV_2LS (rucni ventil sa 2 krajnja prekidaca)                         *)
	(* ======================================================================== *)
	typInHV2LS : STRUCT (* Ulazna struktura FB_HV_2LS. *)
		Enable : BOOL; (* Globalni enable FB-a *)
		CloseFb : BOOL; (* DI - krajnji prekidac ZATVORENO *)
		OpenFb : BOOL; (* DI - krajnji prekidac OTVORENO *)
		ResetAlarm : BOOL; (* Potvrda/resetovanje memorisanog alarma *)
	END_STRUCT;

	typParHV2LS : STRUCT (* Parametarska struktura FB_HV_2LS. *)
		TransitionMaxTime : TIME; (* Maksimalno dozvoljeno vreme medjupolozaja pre transition timeout alarma. *)
		BothActiveFilterTime : TIME; (* Debounce vreme za uslov oba krajnja signala aktivna. *)
	END_STRUCT;

	typOutHV2LS : STRUCT (* Izlazna struktura FB_HV_2LS. *)
		Status : BOOL; (* TRUE = FB je omogucen i konfiguracija je validna. *)
		State : USINT; (* Numericki kod stanja 0-5 *)
		State_comment : STRING[80]; (* Tekstualni opis stanja *)
		AlarmActive : BOOL; (* TRUE = trenutno postoji aktivan alarm uslov. *)
		AlarmLatched : BOOL; (* TRUE = memorisan alarm koji ceka validan reset. *)
		FaultCode : USINT; (* Kod memorisanog alarma. *)
		FaultText : STRING[80]; (* Tekst memorisanog alarma. *)
		Closed : BOOL; (* Fizicka potvrda zatvorenog polozaja: CloseFb=1 i OpenFb=0. *)
		Opened : BOOL; (* Fizicka potvrda otvorenog polozaja: OpenFb=1 i CloseFb=0. *)
		Intermediate : BOOL; (* Fizicki medjupolozaj: OpenFb=0 i CloseFb=0. *)
		FeedbackConflict : BOOL; (* Fizicki konflikt: OpenFb=1 i CloseFb=1. *)
		PositionValid : BOOL; (* TRUE kada je aktivan tacno jedan krajnji signal. *)
		ResetAllowed : BOOL; (* TRUE kada je reset dozvoljen po validnoj reset politici. *)
		ConfigValid : BOOL; (* TRUE kada su vremenski parametri validni. *)
		ConfigFaultText : STRING[80]; (* Tekst prve nevalidne konfiguracione vrednosti. *)
		ActiveConditionCode : USINT; (* Kod trenutno aktivnog uslova (real-time). *)
		Diag : STRING[80]; (* Kratak operativni opis stanja i alarma za HMI. *)
	END_STRUCT;

	typIntHV2LS : STRUCT (* Interna radna struktura FB_HV_2LS. *)
		FaultLatched : BOOL; (* Memorisan alarm do validnog reset-a *)
		FaultCondition : BOOL; (* Trenutni fault uslov u ovom scan-u *)
		ConfigValid : BOOL; (* FALSE kada je parametarska konfiguracija nevalidna. *)
		ConfigFaultText : STRING[80]; (* Opis prve detektovane konfiguracione greske. *)
		FaultCode : USINT; (* Interni broj greske *)
		ActiveConditionCode : USINT; (* Trenutni aktivni uslov za dijagnostiku u realnom vremenu. *)
		ResetAllowed : BOOL; (* Interna memorija dozvole reseta. *)
		Step : USINT; (* Interno stanje *)
		BothActiveRaw : BOOL; (* Sirovi uslov: oba DI aktivna *)
		TransitionRaw : BOOL; (* Sirovi uslov: ni jedan DI aktivan *)
		TonTransition : TON; (* Tajmer za tranziciju - predugo u medjupolozaju *)
		TonBothActive : TON; (* Tajmer za debounce oba signala aktivna *)
	END_STRUCT;

	typCfgHV2LS : STRUCT (* Konfiguraciona struktura konstanti FB_HV_2LS. *)
		T_OpenClose_Valid : TIME; (* Validirano vreme tranzicije *)
		T_BothActive_Valid : TIME; (* Validirano debounce vreme za oba signala *)
		ST_DISABLED : USINT := 0; (* Blok neaktivan *)
		ST_CLOSED : USINT := 1; (* Aktivan - zatvoren *)
		ST_OPEN : USINT := 2; (* Aktivan - otvoren *)
		ST_TRANSITION : USINT := 3; (* Aktivan - u tranziciji *)
		ST_FLT_TRANSITION_TIMEOUT : USINT := 4; (* Medjupolozaj predugo traje (aktivan timeout uslov). *)
		ST_FLT_BOTH_ACTIVE : USINT := 5; (* Oba krajnja signala su aktivna (konflikt feedback-a). *)
		FLT_NONE : USINT := 0; (* Nema aktivnog fault-a *)
		FLT_TRANSITION_TIMEOUT : USINT := 1; (* Predugo u medjupolozaju *)
		FLT_BOTH_ACTIVE : USINT := 2; (* Oba krajnja prekidaca aktivna *)
		FLT_CONFIG_INVALID : USINT := 3; (* Nevalidna konfiguracija vremenskih parametara. *)
		ACT_NONE : USINT := 0; (* Trenutno nema aktivnog alarm uslova. *)
		ACT_TRANSITION_TIMEOUT : USINT := 1; (* Trenutno je aktivan timeout medjupolozaja. *)
		ACT_BOTH_ACTIVE : USINT := 2; (* Trenutno je aktivan uslov oba signala. *)
		ACT_CONFIG_INVALID : USINT := 3; (* Konfiguracija je trenutno nevalidna. *)
	END_STRUCT;

	typHV2LS : STRUCT (* Agregatna struktura svih sekcija za FB_HV_2LS. *)
		Input : typInHV2LS; (* Ulazni signali i komande bloka. *)
		Param : typParHV2LS; (* Parametri vremena i ponasanja. *)
		Output : typOutHV2LS; (* Izlazi, status i dijagnostika. *)
		Internal : typIntHV2LS; (* Interna radna memorija i tajmeri. *)
		Cfg : typCfgHV2LS; (* Konstante state/fault kodova i validirana vremena. *)
	END_STRUCT;

	(* ======================================================================== *)
	(* EH_Flow / FB_EH                                                          *)
	(* ======================================================================== *)
	EH_input : STRUCT (* Ulazna struktura FB_EH_Flow. *)
		Enable : BOOL; (* Omogucavanje grejaca *)
		Setpoint : REAL; (* Zeljena temperatura (degC) *)
		TempIn : REAL; (* Ulazna temperatura (degC) *)
		TempOut : REAL; (* Izlazna temperatura (degC) *)
		FlowSwitch : BOOL; (* Prekidac protoka (TRUE ako ima protoka) *)
		FlowRate : REAL; (* Protok (l/s) *)
		BreakerFB : BOOL; (* Feedback od glavnog prekidaca *)
	END_STRUCT;

	EH_param : STRUCT (* Parametarska struktura FB_EH_Flow. *)
		FlowNominal : REAL; (* Nominalni protok (l/s) *)
		HeaterPower : REAL; (* Snaga pojedinacnog grejaca (kW) *)
		NumHeaters : INT; (* Broj ugradjenih grejaca *)
		ActiveFlowSwitch : BOOL; (* Aktivan flow switch *)
		ActiveFlowMeter : BOOL; (* Aktivan protokomer *)
		OutputType : INT; (* Tip izlaza: 0=analog, 1=PWM *)
		PWM_Width : REAL; (* Sirina PWM-a u sekundama *)
		AnalogMin : INT; (* Raw out min za analog *)
		AnalogMax : INT; (* Raw out max za analog *)
		ScanTime : REAL; (* Vreme skena u sekundama *)
	END_STRUCT;

	EH_output : STRUCT (* Izlazna struktura FB_EH_Flow. *)
		HeaterOn : ARRAY[0..29] OF BOOL; (* Stanje grejaca (TRUE=ON) *)
		AnalogOut : INT; (* Analogni izlaz (skaliran) *)
		PWMOut : REAL; (* PWM izlaz (0-1 duty cycle) *)
		Alarm : BOOL; (* Alarm (TRUE=alarm) *)
		PowerConsumption : REAL; (* Potrosnja energije (kW) *)
		Status : INT; (* Status FB-a: 0=RUNNING, 1=ALARM_OR_WAIT, 2=DISABLED *)
		State : USINT; (* Standardni numericki kod stanja FB-a za HMI *)
		State_comment : STRING[80]; (* Standardni tekstualni opis stanja FB-a *)
		StatusText : STRING[20]; (* Jednoznacan tekstualni opis trenutnog stanja FB-a *)
		OutputTypeText : STRING[12]; (* Tekstualni opis tipa izlaza *)
		AlarmCauseText : STRING[24]; (* Jednoznacan uzrok alarma/neaktivnosti *)
		MainBreaker : BOOL; (* Komanda glavnog prekidaca *)
		ConfigValid : BOOL; (* TRUE kada je izlazna i procesna konfiguracija validna. *)
		ConfigFaultText : STRING[80]; (* Opis prve detektovane nevalidne konfiguracije. *)
	END_STRUCT;

	EH_internal : STRUCT (* Interna radna struktura FB_EH_Flow. *)
		PID_Controller : MTBasicsPID; (* PID kontroler *)
		Temp_Filter : MTFilterMovingAverage; (* Filter za temperaturu *)
		Prev_Enable : BOOL; (* Prethodno stanje Enable *)
		Demand_Percent : REAL; (* Potreba u procentima (0-100%) *)
		Timer_No_Flow : TON; (* Tajmer za nedostatak protoka *)
		Timer_Over_Temp : TON; (* Tajmer za previsoku temperaturu *)
		i : INT; (* Pomocna promenljiva za petlje *)
		Phase : REAL := 0.0; (* Faza za PWM *)
		local_phase : REAL; (* Lokalna faza za grejac *)
		Timer_Breaker_On : TON; (* Tajmer za ukljucivanje *)
		Timer_Breaker_Off : TON; (* Tajmer za iskljucivanje *)
		Breaker_On : BOOL := FALSE; (* Stanje sekvence *)
		Trig_Enable : R_TRIG; (* Rising edge za Enable *)
		Trig_BreakerFB_Fall : F_TRIG; (* Falling edge za BreakerFB *)
		Fault_Latched : BOOL := FALSE; (* Havarijski latch *)
		PID_Init_Pending : BOOL := FALSE; (* Pending reset integratora PID *)
		Filter_Init_Pending : BOOL := FALSE; (* Pending update filtera *)
		NumHeaters_Valid : INT; (* Broj grejaca ogranicen na opseg 0..MAX_HEATERS *)
		ConfigValid : BOOL; (* FALSE kada izlazna ili procesna konfiguracija nije validna. *)
		ConfigFaultText : STRING[80]; (* Tekst prve nevalidne konfiguracije. *)
	END_STRUCT;

	EH_constant : STRUCT (* Struktura konstanti i limita FB_EH_Flow. *)
		MAX_HEATERS : INT := 30; (* Maksimalan broj grejaca *)
		PID_MAX_OUT : REAL := 100.0; (* Maksimalni izlaz PID-a (%) *)
		PID_MIN_OUT : REAL := 0.0; (* Minimalni izlaz PID-a (%) *)
		PID_GAIN : REAL := 1.0; (* Pojacanje PID-a *)
		PID_INTEGRATION_TIME : REAL := 60.0; (* Vreme integracije (s) *)
		PID_DERIVATIVE_TIME : REAL := 0.0; (* Vreme derivacije (s) *)
		FILTER_LENGTH : UINT := 10; (* Duzina filtera *)
		NO_FLOW_TIMEOUT : TIME := T#10s; (* Tajmaut za nedostatak protoka *)
		OVER_TEMP_TIMEOUT : TIME := T#5s; (* Tajmaut za previsoku temp *)
		MAX_TEMP : REAL := 100.0; (* Maksimalna dozvoljena temp (degC) *)
		MIN_FLOW : REAL := 0.1; (* Minimalni protok (l/s) *)
		BREAKER_DELAY : TIME := T#2s; (* Kasnjenje za sekvencu *)
		STATUS_RUNNING : INT := 0; (* Aktivan rad bez alarma *)
		STATUS_ALARM_OR_WAIT : INT := 1; (* Alarm ili cekanje uslova za rad *)
		STATUS_DISABLED : INT := 2; (* Blok onemogucen *)
	END_STRUCT;

	EH_Type : STRUCT (* Agregatna struktura svih sekcija za FB_EH_Flow. *)
		Input : EH_input; (* Ulazi grejaca, temperature i protok. *)
		Param : EH_param; (* Parametri regulacije i tipa izlaza. *)
		Output : EH_output; (* Izlazi, status i alarm indikacije. *)
		Internal : EH_internal; (* Interna stanja regulacije i sekvenci. *)
		Constant : EH_constant; (* Konstante limita i status kodova. *)
	END_STRUCT;

	(* ======================================================================== *)
	(* FB_Pv_AI_AO (zajednicki type-ovi za FAST i SLOW varijantu)              *)
	(* ======================================================================== *)
	typInPvAiAo : STRUCT (* Ulazna struktura FB_Pv_AI_AO (FAST/SLOW). *)
		Enable : BOOL; (* Globalna dozvola rada bloka. FALSE gasi izlaz i tracking. *)
		Reset : BOOL; (* Reset fault stanja i internih tajmera/nadzora. *)
		EnableManual : BOOL; (* TRUE = koristi ManualValue_Percent, FALSE = koristi SP_Percent. *)
		ForceCmd : BOOL; (* TRUE = dozvoli prolaz komande i kada je fault aktivan. *)
		AI_Raw : INT; (* Sirova AI vrednost ventila u opsegu 0..32767. *)
		SP_Percent : REAL; (* Auto zadavanje ventila u procentima 0.0..100.0. *)
		ManualValue_Percent : REAL; (* Manuelno zadavanje ventila u procentima 0.0..100.0. *)
	END_STRUCT;

	typParPvAiAo : STRUCT (* Parametarska struktura FB_Pv_AI_AO (FAST/SLOW). *)
		HoldOutputOnFault : BOOL; (* TRUE = na fault drzi poslednji validan izlaz; FALSE = izlaz ide na 0%. *)
		DeviationOnLimit : REAL; (* Prag (%): ulazak u devijantno stanje. *)
		DeviationOffLimit : REAL; (* Prag (%): izlazak iz devijantnog stanja (histereza). *)
		DeviationTime : TIME; (* Maksimalno dozvoljeno trajanje devijacije pre fault-a. *)
	END_STRUCT;

	typOutPvAiAo : STRUCT (* Izlazna struktura FB_Pv_AI_AO (FAST/SLOW). *)
		PV_Percent : REAL; (* Skalirana procesna vrednost ventila u %. *)
		ActiveSP_Percent : REAL; (* Aktivna komanda (auto/manual) koja upravlja izlazom. *)
		AppliedOutput_Percent : REAL; (* Stvarno primenjena izlazna komanda nakon fault logike. *)
		FrozenOutput_Percent : REAL; (* Poslednja validna komanda za hold-on-fault scenario. *)
		AO_Raw : INT; (* Skalirani AO izlaz u opsegu 0..32767. *)
		DeviationPercent : REAL; (* ABS(ActiveSP - PV) u procentima. *)
		InDeviation : BOOL; (* TRUE kada je aktivno devijantno stanje. *)
		InTolerance : BOOL; (* TRUE kada je devijacija unutar DeviationOff granice. *)
		DeviationTimeout : BOOL; (* TRUE kada je devijacija trajala duze od dozvoljenog vremena. *)
		FaultActive : BOOL; (* Latched fault status bloka. *)
		ManualActive : BOOL; (* Informativno: aktivan manuelni mod. *)
		ForceActive : BOOL; (* Informativno: ForceCmd trenutno premostava fault blokadu. *)
		CommandPermitted : BOOL; (* TRUE kada komanda sme direktno na izlaz. *)
		Valid : BOOL; (* Informativno: blok je omogucen (Enable=TRUE). *)
		AI_Raw_Limited : INT; (* Ogranicena AI vrednost 0..32767. *)
		SP_Percent_Limited : REAL; (* Ogranicen auto SP 0.0..100.0. *)
		ManualValue_Limited : REAL; (* Ogranicen manuelni SP 0.0..100.0. *)
		ActiveSP_Limited : REAL; (* Ogranicena aktivna komanda 0.0..100.0. *)
		AppliedOutput_Limited : REAL; (* Ogranicena primenjena komanda 0.0..100.0. *)
		DeviationOn_Limited : REAL; (* Ogranicen prag ulaska u devijaciju. *)
		DeviationOff_Limited : REAL; (* Ogranicen prag izlaska iz devijacije. *)
		DeviationTime_Effective : TIME; (* Efektivno vreme devijacije nakon validacije parametra. *)
		DeviationElapsed : TIME; (* Proteklo vreme aktivne devijacije (ET iz tajmera). *)
		Status : BOOL; (* Standardni status: TRUE u normalnom radu bez fault-a. *)
		State : USINT; (* Standardni numericki kod stanja za HMI/SCADA. *)
		State_comment : STRING[80]; (* Standardni tekst opisa stanja. *)
	END_STRUCT;

	typIntPvAiAo : STRUCT (* Interna struktura FAST varijante FB_Pv_AI_AO. *)
		rAi : REAL; (* Pomocna REAL promenljiva za AI->% skaliranje. *)
		rAo : REAL; (* Pomocna REAL promenljiva za %->AO skaliranje. *)
		AO_Raw_Calc : INT; (* Interno izracunata AO raw vrednost pre ogranicenja. *)
		FB_DeviationTimer : TON; (* Tajmer trajanja devijantnog stanja. *)
	END_STRUCT;

	typIntPvAiAoSlow : STRUCT (* Interna struktura SLOW varijante FB_Pv_AI_AO. *)
		rAi : REAL; (* Pomocna REAL promenljiva za AI->% skaliranje. *)
		rAo : REAL; (* Pomocna REAL promenljiva za %->AO skaliranje. *)
		AO_Raw_Calc : INT; (* Interno izracunata AO raw vrednost pre ogranicenja. *)
		FB_DeviationTimer : TON; (* Tajmer trajanja devijantnog stanja. *)
		TrackTimer : TON; (* Glavni tajmer maksimalnog trajanja aktivnog poteza (Tmax). *)
		StartMoveTimer : TON; (* Tajmer cekanja inicijalnog pomeranja nakon komande. *)
		DirectionTimer : TON; (* Tajmer potvrde pogresnog smera kretanja. *)
		StallTimer : TON; (* Tajmer zastoja ventila tokom aktivnog poteza. *)
		TrackActive : BOOL; (* TRUE dok je aktivan nadzor jednog poteza ventila. *)
		TrackDirectionOpen : BOOL; (* TRUE = ocekuje se otvaranje (rast PV); FALSE = zatvaranje. *)
		MovementStarted : BOOL; (* TRUE kada je detektovano pocetno pomeranje posle komande. *)
		FaultReasonText : STRING[80]; (* Tekstualni uzrok fault-a za State_comment. *)
		PrevSP : REAL; (* Aktivni SP iz prethodnog ciklusa, za detekciju koraka. *)
		PrevPV : REAL; (* PV iz prethodnog ciklusa, za detekciju trenda/smera. *)
		PV_AtTrackStart : REAL; (* PV vrednost u trenutku starta poteza. *)
		LastProgressPV : REAL; (* Poslednja PV referenca za procenu progresa/stalla. *)
		StepDeltaPercent : REAL; (* Velicina koraka komande u %, ABS(NewSP-PrevSP). *)
		ExpectedTravelSec : REAL; (* Ocekivano vreme poteza u sekundama po velicini koraka. *)
		TminSec : REAL; (* Donja granica dozvoljenog vremena poteza. *)
		TmaxSec : REAL; (* Gornja granica dozvoljenog vremena poteza. *)
		ActualTravelSec : REAL; (* Stvarno ostvareno vreme poteza pri zavrsetku. *)
		TravelTimeOpenFull : TIME := T#120s; (* Puno vreme otvaranja 0->100%. *)
		TravelTimeCloseFull : TIME := T#120s; (* Puno vreme zatvaranja 100->0%. *)
		TimeTolerancePercent : REAL := 30.0; (* Dozvoljeno vremensko odstupanje oko Texp. *)
		StartMoveTimeout : TIME := T#5s; (* Max cekanje da ventil krene nakon nove komande. *)
		DirectionCheckTime : TIME := T#5s; (* Potvrda pogresnog smera ako traje duze od ovog vremena. *)
		StallTimeout : TIME := T#15s; (* Max dozvoljen zastoj tokom aktivnog kretanja. *)
		MovementStartDeltaPercent : REAL := 0.5; (* Minimalna promena PV (%) za potvrdu da je kretanje pocelo. *)
		PerScanProgressMinPercent : REAL := 0.05; (* Minimalni progres po ciklusu za izbegavanje stall detekcije. *)
		DirectionEpsPercent : REAL := 0.02; (* Mrtva zona za proveru smera da se filtrira sum. *)
		EnableTooFastFault : BOOL := FALSE; (* TRUE = prebrz potez tretirati kao fault, FALSE = samo info. *)
	END_STRUCT;

	typConstPvAiAo : STRUCT (* Struktura konstanti i state kodova FB_Pv_AI_AO. *)
		RAW_MIN : INT := 0; (* Donja granica sirovog AI/AO opsega. *)
		RAW_MAX : INT := 32767; (* Gornja granica sirovog AI/AO opsega. *)
		PCT_MIN : REAL := 0.0; (* Donja granica procentualnog opsega. *)
		PCT_MAX : REAL := 100.0; (* Gornja granica procentualnog opsega. *)
		MIN_DEV_TIME : TIME := T#1ms; (* Minimalno efektivno vreme devijacije. *)
		REC_DEV_ON_LIMIT : REAL := 8.0; (* Preporucen prag ulaska u devijaciju za commissioning. *)
		REC_DEV_OFF_LIMIT : REAL := 3.0; (* Preporucen prag izlaska iz devijacije za commissioning. *)
		REC_DEV_TIME : TIME := T#5s; (* Preporuceno vreme potvrde devijacije za commissioning. *)
		ST_DISABLED : USINT := 0; (* Blok nije omogucen. *)
		ST_AUTO_ACTIVE : USINT := 1; (* Normalan auto rad. *)
		ST_MANUAL_ACTIVE : USINT := 2; (* Normalan manual rad. *)
		ST_DEVIATION_ACTIVE : USINT := 3; (* Aktivno pracenje devijacije. *)
		ST_FAULT_HOLD : USINT := 4; (* Fault aktivan, izlaz hold/zero. *)
		ST_FAULT_FORCE : USINT := 5; (* Fault aktivan, ali ForceCmd dozvoljava komandu. *)
	END_STRUCT;

	typPvAiAo : STRUCT (* Agregatna struktura svih sekcija za FB_Pv_AI_AO. *)
		Input : typInPvAiAo; (* Ulazni procesni i upravljacki signali. *)
		Param : typParPvAiAo; (* Parametri ponasanja i pragovi logike. *)
		Output : typOutPvAiAo; (* Izlazi, statusi i dijagnostika bloka. *)
		Internal : typIntPvAiAo; (* Interne pomocne promenljive i tajmeri. *)
		Constant : typConstPvAiAo; (* Konstante granica, state kodovi i preporuke. *)
	END_STRUCT;

	(* ======================================================================== *)
	(* FB_PV_AO_NO_FB (proporcionalni ventil bez pozicionog feedback-a)  *)
	(* ======================================================================== *)
	typInPvAoNoFb : STRUCT (* Ulazna struktura FB_PV_AO_NO_FB. *)
		Enable : BOOL; (* Globalna dozvola rada bloka. *)
		AutoSP : REAL; (* Auto zadavanje u procentima. *)
		ManualMode : BOOL; (* TRUE = aktivan manuelni rezim. *)
		ManualOut : REAL; (* Manuelna izlazna komanda u procentima. *)
		ForceCmd : BOOL; (* TRUE = dozvola izlaza i kada je fault aktivan. *)
		ResetFault : BOOL; (* Reset latched fault stanja. *)
	END_STRUCT;

	typParPvAoNoFb : STRUCT (* Parametarska struktura FB_PV_AO_NO_FB. *)
		OutMin : REAL; (* Donja granica dozvoljenog izlaza u %. *)
		OutMax : REAL; (* Gornja granica dozvoljenog izlaza u %. *)
		RampUp : REAL; (* Maksimalni porast izlaza po ciklusu u %. *)
		RampDown : REAL; (* Maksimalni pad izlaza po ciklusu u %. *)
		OnDelay : TIME; (* Kasnjenje aktivacije izlaza iznad OutMin. *)
		OffDelay : TIME; (* Kasnjenje vracanja izlaza na OutMin. *)
		HoldOnFault : BOOL; (* TRUE = drzi poslednji validan izlaz na fault-u. *)
	END_STRUCT;

	typOutPvAoNoFb : STRUCT (* Izlazna struktura FB_PV_AO_NO_FB. *)
		AO_Cmd : REAL; (* Finalna komandna vrednost ventila u %. *)
		Status : BOOL; (* Standardni status: TRUE kada nema fault-a i Enable=TRUE. *)
		State : USINT; (* Standardni numericki kod stanja. *)
		State_comment : STRING[80]; (* Tekstualni opis stanja. *)
		FaultActive : BOOL; (* Latched fault status bloka. *)
		FaultCode : USINT; (* Numericki kod fault-a. *)
		ManualActive : BOOL; (* Informativno: manuelni rezim je aktivan. *)
		ForceActive : BOOL; (* Informativno: ForceCmd trenutno premostava fault. *)
		CmdTarget : REAL; (* Izabrana komanda pre delay/ramp obrade. *)
		CmdLimited : REAL; (* Komanda ogranicena na OutMin..OutMax. *)
		CmdDelayed : REAL; (* Komanda nakon OnDelay/OffDelay obrade. *)
		ParamInvalid : BOOL; (* TRUE kada je konfiguracija parametara nevalidna. *)
		OutMin_Effective : REAL; (* Efektivna donja granica posle validacije. *)
		OutMax_Effective : REAL; (* Efektivna gornja granica posle validacije. *)
		RampUp_Effective : REAL; (* Efektivni maksimalni porast komande po ciklusu. *)
		RampDown_Effective : REAL; (* Efektivni maksimalni pad komande po ciklusu. *)
		OnDelay_Effective : TIME; (* Efektivno kasnjenje aktivacije komande. *)
		OffDelay_Effective : TIME; (* Efektivno kasnjenje deaktivacije komande. *)
	END_STRUCT;

	typIntPvAoNoFb : STRUCT (* Interna radna struktura FB_PV_AO_NO_FB. *)
		CmdWorking : REAL; (* Interna radna komanda posle delay i ramp logike. *)
		LastHealthyCmd : REAL; (* Poslednja validna komanda bez fault-a. *)
		RiseRequest : BOOL; (* Zahtev za izlaz iznad OutMin. *)
		FallRequest : BOOL; (* Zahtev za izlaz na OutMin. *)
		OnDelayTimer : TON; (* Tajmer kasnjenja aktivacije komande. *)
		OffDelayTimer : TON; (* Tajmer kasnjenja deaktivacije komande. *)
		EpsPercent : REAL := 0.001; (* Mrtva zona za porejenje realnih vrednosti. *)
	END_STRUCT;

	typConstPvAoNoFb : STRUCT (* Struktura konstanti i state/fault kodova FB_PV_AO_NO_FB. *)
		PCT_MIN : REAL := 0.0; (* Donja granica procentualnog opsega izlaza. *)
		PCT_MAX : REAL := 100.0; (* Gornja granica procentualnog opsega izlaza. *)
		STEP_MIN : REAL := 0.0001; (* Minimalan pozitivan korak za ramp validaciju. *)
		FLT_NONE : USINT := 0; (* Nema aktivnog fault-a. *)
		FLT_PARAM_INVALID : USINT := 1; (* Parametri bloka nisu validni. *)
		ST_DISABLED : USINT := 0; (* Blok nije omogucen. *)
		ST_AUTO_ACTIVE : USINT := 1; (* Auto rezim aktivan bez fault-a. *)
		ST_MANUAL_ACTIVE : USINT := 2; (* Manual rezim aktivan bez fault-a. *)
		ST_FAULT_HOLD : USINT := 3; (* Fault aktivan i izlaz je hold/bez komande. *)
		ST_FAULT_FORCE : USINT := 4; (* Fault aktivan uz ForceCmd premoscenje. *)
	END_STRUCT;

	typPvAoNoFb : STRUCT (* Agregatna struktura svih sekcija za FB_PV_AO_NO_FB. *)
		Input : typInPvAoNoFb; (* Ulazi komandi i servisnih signala bloka. *)
		Param : typParPvAoNoFb; (* Parametri granica, rampi i fault logike. *)
		Output : typOutPvAoNoFb; (* Izlazi komande, status i dijagnostika. *)
		Internal : typIntPvAoNoFb; (* Interna radna stanja i tajmeri. *)
		Constant : typConstPvAoNoFb; (* Konstante limita, state i fault kodova. *)
	END_STRUCT;

	(* ======================================================================== *)
	(* FB_AirRelease (odzracivanje cevovoda sa 1 do 3 LS senzora)              *)
	(* ======================================================================== *)
	typInAirRelease : STRUCT (* Ulazna struktura FB_AirRelease. *)
		Enable : BOOL; (* Spoljna dozvola automatskog odzracivanja; FALSE pokrece bezbedno zatvaranje ventila. *)
		EnableManual : BOOL; (* TRUE = direktna rucna komanda ventila ima prioritet nad automatskom pressure/LS logikom. *)
		ManualSP_Percent : REAL; (* Direktna rucna komanda proporcionalnog ventila [%]; ogranicava se na 0.0..100.0. *)
		Pressure_bar : REAL; (* Skalirani pritisak nadziranog cevovoda [bar]; ocekovani radni opseg >= 0.0 bar. *)
		LS1_Upper : BOOL; (* Gornji i obavezni LS1; TRUE = voda potvrdena na najvisoj mernoj tacki. *)
		LS2_Middle : BOOL; (* Drugi LS odozgo; koristi se samo kada je NumberOfLS >= 2; TRUE = voda prisutna. *)
		LS3_Lower : BOOL; (* Treci i najnizi LS; koristi se samo kada je NumberOfLS = 3; TRUE = voda prisutna. *)
		ResetAlarm : BOOL; (* Impuls za reset memorisanog alarma kada vise nema aktivnog alarmnog uslova. *)
	END_STRUCT;

	typParAirReleaseStage : STRUCT (* Parametri jednog LS stepena odzracivanja. *)
		SP_Percent : REAL; (* Pocetna/granicna komanda pripadajuceg LS stepena [%]; dozvoljeno 0.0..100.0. *)
		Ramp_PercentPerSecond : REAL; (* Ista rampa otvaranja i zatvaranja stepena [%/s]; mora biti > 0.0. *)
		ConfirmTime_s : REAL; (* Neprekidno vreme potvrde aktivacije i deaktivacije LS signala [s]; dozvoljeno 0.0..3600.0 s. *)
	END_STRUCT;

	typParAirRelease : STRUCT (* Parametarska struktura FB_AirRelease; projekat je deklarise kao RETAIN i menja sa HMI-ja. *)
		NumberOfLS : USINT; (* Broj fizicki ugradenih LS senzora; dozvoljeno 1..3; numeracija je uvek odozgo nadole. *)
		PressureSP_bar : REAL; (* Prag ukljucenja monitoringa aktivnog pritiska [bar]; mora biti >= 0.0. *)
		PressureHysteresis_bar : REAL; (* Histereza iskljucenja pritiska [bar]; opseg 0.0..PressureSP_bar. *)
		LS1 : typParAirReleaseStage; (* Gornji i uvek aktivan stepen. *)
		LS2 : typParAirReleaseStage; (* Srednji stepen za 2/3 LS. *)
		LS3 : typParAirReleaseStage; (* Najnizi stepen samo za 3 LS. *)
	END_STRUCT;

	typOutAirRelease : STRUCT (* Izlazna struktura FB_AirRelease. *)
		ValveSP_Percent : REAL; (* Finalna auto/manual komanda proporcionalnog ventila [%], ogranicena na 0.0..100.0. *)
		Status : BOOL; (* TRUE kada je FB omogucen, konfiguracija validna, vreme ciklusa validno i nema alarma. *)
		State : USINT; (* Numericki kod trenutnog operativnog stanja za HMI i visi nivo. *)
		State_comment : STRING[80]; (* Jednoznacan tekst trenutnog operativnog stanja. *)
		ManualActive : BOOL; (* TRUE kada rucna komanda direktno upravlja izlazom ventila. *)
		PressureActive : BOOL; (* TRUE kada je pritisak presao PressureSP_bar i nije pao ispod SP-histereza. *)
		LS1_Confirmed : BOOL; (* Filtrirano stanje gornjeg LS1 posle ConfirmTime_s. *)
		LS2_Confirmed : BOOL; (* Filtrirano stanje LS2. *)
		LS3_Confirmed : BOOL; (* Filtrirano stanje LS3. *)
		ActiveStage : USINT; (* Aktivni LS stepen komande: 0=manual, 1=LS1, 2=LS2, 3=LS3. *)
		Opening : BOOL; (* TRUE kada se automatska komanda povecava prema SP-u aktivnog stepena. *)
		Closing : BOOL; (* TRUE kada se automatska komanda smanjuje prema 0%. *)
		AlarmActive : BOOL; (* TRUE kada trenutno postoji alarmni uslov. *)
		AlarmLatched : BOOL; (* TRUE kada je memorisan prvi alarm i ceka reset. *)
		FaultCode : USINT; (* Kod prvog memorisanog alarma. *)
		FaultText : STRING[80]; (* Tekst prvog memorisanog alarma. *)
		ActiveConditionCode : USINT; (* Kod trenutno aktivnog alarmnog uslova. *)
		ResetAllowed : BOOL; (* TRUE kada je dozvoljen reset memorisanog alarma. *)
		ConfigValid : BOOL; (* TRUE kada su svi aktivni parametri validni. *)
		ConfigFaultText : STRING[80]; (* Opis prve nevalidne parametarske vrednosti. *)
		LSSequenceInvalid : BOOL; (* TRUE kada potvrdeni LS redosled nije fizicki moguc. *)
		CycleTime_s : REAL; (* Izmereno vreme task ciklusa [s]. *)
		Diag : STRING[80]; (* Kratak operativni opis za HMI. *)
	END_STRUCT;

	typIntAirRelease : STRUCT (* Interna radna struktura FB_AirRelease. *)
		RtInfo : RTInfo; (* B&R runtime informacija za stvarno vreme task ciklusa. *)
		ConfigValid : BOOL;
		RuntimeTimeValid : BOOL;
		ConfigFaultText : STRING[80];
		PressureActive : BOOL;
		ControlActivePrev : BOOL;
		LS1Confirmed : BOOL;
		LS2Confirmed : BOOL;
		LS3Confirmed : BOOL;
		LS1ConfirmedPrev : BOOL;
		LS2ConfirmedPrev : BOOL;
		LS3ConfirmedPrev : BOOL;
		TonLS1Change : TON;
		TonLS2Change : TON;
		TonLS3Change : TON;
		LS1ConfirmTime : TIME;
		LS2ConfirmTime : TIME;
		LS3ConfirmTime : TIME;
		ValveCmd : REAL;
		TargetSP : REAL;
		ActiveRamp : REAL;
		RampStep : REAL;
		ActiveStage : USINT;
		OpeningMode : BOOL;
		LSSequenceInvalid : BOOL;
		FaultCondition : BOOL;
		FaultLatched : BOOL;
		FaultCode : USINT;
		ActiveConditionCode : USINT;
		ResetAllowed : BOOL;
		Step : USINT;
	END_STRUCT;

	typConstAirRelease : STRUCT (* Konstante granica, stanja i alarma FB_AirRelease. *)
		PCT_MIN : REAL := 0.0;
		PCT_MAX : REAL := 100.0;
		RAMP_MIN : REAL := 0.0001;
		CONFIRM_TIME_MAX_S : REAL := 3600.0;
		CYCLE_TIME_MAX_S : REAL := 1.0;
		SAFE_CLOSE_SP : REAL := 20.0;
		SAFE_CLOSE_RAMP : REAL := 2.0;
		ST_DISABLED : USINT := 0;
		ST_WAIT_PRESSURE : USINT := 1;
		ST_OPENING_LS1 : USINT := 2;
		ST_OPENING_LS2 : USINT := 3;
		ST_OPENING_LS3 : USINT := 4;
		ST_CLOSING_LS1 : USINT := 5;
		ST_CLOSING_LS2 : USINT := 6;
		ST_CLOSED : USINT := 7;
		ST_FAULT_SAFE_CLOSE : USINT := 8;
		ST_MANUAL : USINT := 9;
		FLT_NONE : USINT := 0;
		FLT_CONFIG_INVALID : USINT := 1;
		FLT_LS_SEQUENCE_INVALID : USINT := 2;
		FLT_RUNTIME_TIME_INVALID : USINT := 3;
		ACT_NONE : USINT := 0;
		ACT_CONFIG_INVALID : USINT := 1;
		ACT_LS_SEQUENCE_INVALID : USINT := 2;
		ACT_RUNTIME_TIME_INVALID : USINT := 3;
	END_STRUCT;

	typAirRelease : STRUCT (* Agregatna struktura svih sekcija FB_AirRelease. *)
		Input : typInAirRelease;
		Param : typParAirRelease;
		Output : typOutAirRelease;
		Internal : typIntAirRelease;
		Constant : typConstAirRelease;
	END_STRUCT;
END_TYPE
```

#### BR_Lib.fun - Exported functions and function blocks
```iecst
(* ============================================================================ *)
(* BR_LIB - SVE FB VAR DEKLARACIJE (B&R Automation Studio stil)                *)
(* Sadrzi samo deklaracije interfejsa i internih varijabli po FUNCTION_BLOCK-u. *)
(* Bez implementacione logike.                                                  *)
(* ============================================================================ *)

FUNCTION_BLOCK FBAI01_DI01 (* Skaliranje transmitera sa AI + statusnim DI signalom *) (*$GROUP=User,$CAT=User,$GROUPICON=User.png,$CATICON=User.png*) (* Deklaracija interfejsa FUNCTION_BLOCK FBAI01_DI01. *)
VAR_INPUT
	AI_Input : typInAI01_DI01; (* Deklaracija ulazne strukture bloka FBAI01_DI01. *)
	AI_Param : typParAI01_DI01; (* Deklaracija parametarske strukture bloka FBAI01_DI01. *)
END_VAR
VAR_OUTPUT
	AI_Output : typOutAI01_DI01; (* Deklaracija izlazne strukture bloka FBAI01_DI01. *)
END_VAR
VAR
	AI_Internal : typIntAI01_DI01; (* Deklaracija interne strukture bloka FBAI01_DI01. *)
	AI_Constant : typConstAI01_DI01; (* Deklaracija strukture konstanti bloka FBAI01_DI01. *)
END_VAR
END_FUNCTION_BLOCK

FUNCTION_BLOCK FBAI01_DI01_DO02 (* Skaliranje transmitera sa AI + status DI + 2 DO izbora opsega *) (*$GROUP=User,$CAT=User,$GROUPICON=User.png,$CATICON=User.png*) (* Deklaracija interfejsa FUNCTION_BLOCK FBAI01_DI01_DO02. *)
VAR_INPUT
	AI_Input : typInAI01_DI01_DO02; (* Deklaracija ulazne strukture bloka FBAI01_DI01_DO02. *)
	AI_Param : typParAI01_DI01_DO02; (* Deklaracija parametarske strukture bloka FBAI01_DI01_DO02. *)
END_VAR
VAR_OUTPUT
	AI_Output : typOutAI01_DI01_DO02; (* Deklaracija izlazne strukture bloka FBAI01_DI01_DO02. *)
END_VAR
VAR
	AI_Internal : typIntAI01_DI01_DO02; (* Deklaracija interne strukture bloka FBAI01_DI01_DO02. *)
	AI_Constant : typConstAI01_DI01_DO02; (* Deklaracija strukture konstanti bloka FBAI01_DI01_DO02. *)
END_VAR
END_FUNCTION_BLOCK

FUNCTION_BLOCK FB_DI (* Univerzalni DI sa opcionim status signalom i fault dijagnostikom *) (*$GROUP=User,$CAT=User,$GROUPICON=User.png,$CATICON=User.png*) (* Deklaracija interfejsa FUNCTION_BLOCK FB_DI. *)
VAR_INPUT
	DI_Input : typInDI; (* Deklaracija ulazne strukture bloka FB_DI. *)
	DI_Param : typParDI; (* Deklaracija parametarske strukture bloka FB_DI. *)
END_VAR
VAR_OUTPUT
	DI_Output : typOutDI; (* Deklaracija izlazne strukture bloka FB_DI. *)
END_VAR
VAR
	DI_Internal : typIntDI; (* Deklaracija interne strukture bloka FB_DI. *)
	DI_Constant : typConstDI; (* Deklaracija strukture konstanti bloka FB_DI. *)
END_VAR
END_FUNCTION_BLOCK

FUNCTION_BLOCK FB_V_ON_OFF_FB (* Predlog FB za ON/OFF ventil - odvojeno od FB_AI_01 *) (* Deklaracija interfejsa FUNCTION_BLOCK FB_V_ON_OFF_FB. *)
VAR_INPUT
	Open : BOOL; (* Komandni zahtev: TRUE otvori, FALSE zatvori *)
	V_Input : typInVOnOff; (* Deklaracija ulazne strukture bloka FB_V_ON_OFF_FB. *)
	V_Param : typParVOnOff := (
		DeEnergizedOpen := FALSE,
		FbOpenExists := TRUE,
		FbCloseExists := TRUE,
		OpenMinTime := T#1s,
		OpenMaxTime := T#30s,
		CloseMinTime := T#1s,
		CloseMaxTime := T#30s,
		StableFbDelay := T#2s
	);
END_VAR
VAR_OUTPUT
	Opened : BOOL; (* Otvoren polozaj koji FB koristi: fizicki potvrdjen ili vremenski pretpostavljen. *)
	Closed : BOOL; (* Zatvoren polozaj koji FB koristi: fizicki potvrdjen ili vremenski pretpostavljen. *)
	V_Output : typOutVOnOff; (* Deklaracija izlazne strukture bloka FB_V_ON_OFF_FB. *)
END_VAR
VAR
	Internal : typIntVOnOff; (* Deklaracija interne strukture bloka FB_V_ON_OFF_FB. *)
	Cfg : typCfgVOnOff; (* Deklaracija konfiguracione strukture bloka FB_V_ON_OFF_FB. *)
END_VAR
END_FUNCTION_BLOCK

FUNCTION_BLOCK FB_V_EMV (* Elektromotorni ventil sa odvojenim OPEN/CLOSE komandama. *) (* Deklaracija interfejsa FUNCTION_BLOCK FB_V_EMV. *)
VAR_INPUT
	Open : BOOL; (* Automatski zahtev polozaja: TRUE = OPEN, FALSE = CLOSE. *)
	V_Input : typInVEmv; (* Deklaracija ulazne strukture bloka FB_V_EMV. *)
	V_Param : typParVEmv := (
		LampOpenExists := TRUE,
		LampCloseExists := TRUE,
		OpenFbExists := TRUE,
		CloseFbExists := TRUE,
		OverTorqueExists := FALSE,
		UnexpectedOpenLimitCheck := FALSE,
		UnexpectedCloseLimitCheck := FALSE,
		OpenMaxTime := T#30s,
		CloseMaxTime := T#30s,
		DeadTime := T#500ms,
		EndLimitFilterTime := T#50ms,
		PositionFbFilterTime := T#100ms,
		OverTorqueFilterTime := T#20ms,
		PositionConfirmTime := T#1s,
		StableFbLossTime := T#0ms
	); (* Parametri konfiguracije, nadzora i filtracije FB_V_EMV. *)
END_VAR
VAR_OUTPUT
	Opened : BOOL; (* Cista fizicka potvrda otvorenog polozaja. *)
	Closed : BOOL; (* Cista fizicka potvrda zatvorenog polozaja. *)
	V_Output : typOutVEmv; (* Deklaracija izlazne strukture bloka FB_V_EMV. *)
END_VAR
VAR
	Internal : typIntVEmv; (* Deklaracija interne strukture bloka FB_V_EMV. *)
	Cfg : typCfgVEmv; (* Deklaracija konfiguracione strukture bloka FB_V_EMV. *)
END_VAR
END_FUNCTION_BLOCK

FUNCTION_BLOCK FB_HV_2LS (* Rucni ventil sa dva krajnja prekidaca *) (*$GROUP=User,$CAT=User,$GROUPICON=User.png,$CATICON=User.png*) (* Deklaracija interfejsa FUNCTION_BLOCK FB_HV_2LS. *)
VAR_INPUT
	HV_Input : typInHV2LS; (* Deklaracija ulazne strukture bloka FB_HV_2LS. *)
	HV_Param : typParHV2LS := (
		TransitionMaxTime := T#30s,
		BothActiveFilterTime := T#500ms
	); (* Deklaracija parametarske strukture bloka FB_HV_2LS. *)
END_VAR
VAR_OUTPUT
	HV_Output : typOutHV2LS; (* Deklaracija izlazne strukture bloka FB_HV_2LS. *)
END_VAR
VAR
	Internal : typIntHV2LS; (* Deklaracija interne strukture bloka FB_HV_2LS. *)
	Cfg : typCfgHV2LS; (* Deklaracija konfiguracione strukture bloka FB_HV_2LS. *)
END_VAR
END_FUNCTION_BLOCK

FUNCTION_BLOCK FB_EH_Flow (*TODO: FB za upravljanje elektricnim grejacima*) (*$GROUP=Pedja,$CAT=User,$GROUPICON=User.png,$CATICON=User.png*) (* Deklaracija interfejsa FUNCTION_BLOCK FB_EH_Flow. *)
VAR_INPUT
	EH_Input : EH_input; (* Deklaracija ulazne strukture bloka FB_EH_Flow. *)
	EH_Param : EH_param; (* Deklaracija parametarske strukture bloka FB_EH_Flow. *)
END_VAR
VAR_OUTPUT
	EH_Output : EH_output; (* Deklaracija izlazne strukture bloka FB_EH_Flow. *)
END_VAR
VAR
	EH_Internal : EH_internal; (* Deklaracija interne strukture bloka FB_EH_Flow. *)
	EH_Constant : EH_constant; (* Deklaracija strukture konstanti bloka FB_EH_Flow. *)
END_VAR
END_FUNCTION_BLOCK

FUNCTION_BLOCK FB_PvAiAo_Fast (* Deklaracija interfejsa FUNCTION_BLOCK FB_PvAiAo_Fast. *)
VAR_INPUT
	PV_Input : typInPvAiAo; (* Deklaracija ulazne strukture bloka FB_PvAiAo_Fast. *)
	PV_Param : typParPvAiAo; (* Deklaracija parametarske strukture bloka FB_PvAiAo_Fast. *)
END_VAR
VAR_OUTPUT
	PV_Output : typOutPvAiAo; (* Deklaracija izlazne strukture bloka FB_PvAiAo_Fast. *)
END_VAR
VAR
	PV_Internal : typIntPvAiAo; (* Deklaracija interne strukture bloka FB_PvAiAo_Fast. *)
	PV_Constant : typConstPvAiAo; (* Deklaracija strukture konstanti bloka FB_PvAiAo_Fast. *)
END_VAR
END_FUNCTION_BLOCK

FUNCTION_BLOCK FB_PvAiAo_Slow (* Deklaracija interfejsa FUNCTION_BLOCK FB_PvAiAo_Slow. *)
VAR_INPUT
	PV_Input : typInPvAiAo; (* Deklaracija ulazne strukture bloka FB_PvAiAo_Slow. *)
	PV_Param : typParPvAiAo; (* Deklaracija parametarske strukture bloka FB_PvAiAo_Slow. *)
END_VAR
VAR_OUTPUT
	PV_Output : typOutPvAiAo; (* Deklaracija izlazne strukture bloka FB_PvAiAo_Slow. *)
END_VAR
VAR
	PV_Internal : typIntPvAiAoSlow; (* Deklaracija interne strukture bloka FB_PvAiAo_Slow. *)
	PV_Constant : typConstPvAiAo; (* Deklaracija strukture konstanti bloka FB_PvAiAo_Slow. *)
END_VAR
END_FUNCTION_BLOCK

FUNCTION_BLOCK FB_PvAoNoFb (* Deklaracija interfejsa FUNCTION_BLOCK FB_PvAoNoFb. *)
VAR_INPUT
	PV_Input : typInPvAoNoFb; (* Deklaracija ulazne strukture bloka FB_PvAoNoFb. *)
	PV_Param : typParPvAoNoFb; (* Deklaracija parametarske strukture bloka FB_PvAoNoFb. *)
END_VAR
VAR_OUTPUT
	PV_Output : typOutPvAoNoFb; (* Deklaracija izlazne strukture bloka FB_PvAoNoFb. *)
END_VAR
VAR
	PV_Internal : typIntPvAoNoFb; (* Deklaracija interne strukture bloka FB_PvAoNoFb. *)
	PV_Constant : typConstPvAoNoFb; (* Deklaracija strukture konstanti bloka FB_PvAoNoFb. *)
END_VAR
END_FUNCTION_BLOCK

FUNCTION_BLOCK FB_AirRelease (* Automatsko i rucno odzracivanje cevovoda sa 1 do 3 LS senzora. *) (*$GROUP=User,$CAT=User,$GROUPICON=User.png,$CATICON=User.png*)
VAR_INPUT
	AR_Input : typInAirRelease; (* Procesni ulazi: Enable, manual komanda, pritisak [bar], LS1..LS3 i reset alarma. *)
	AR_Param : typParAirRelease := (
		NumberOfLS := 1,
		PressureSP_bar := 1.5,
		PressureHysteresis_bar := 0.5,
		LS1 := (SP_Percent := 20.0, Ramp_PercentPerSecond := 2.0, ConfirmTime_s := 1.0),
		LS2 := (SP_Percent := 54.5, Ramp_PercentPerSecond := 8.5, ConfirmTime_s := 1.0),
		LS3 := (SP_Percent := 89.0, Ramp_PercentPerSecond := 15.0, ConfirmTime_s := 1.0)
	);
END_VAR
VAR_OUTPUT
	AR_Output : typOutAirRelease;
END_VAR
VAR
	AR_Internal : typIntAirRelease;
	AR_Constant : typConstAirRelease;
END_VAR
END_FUNCTION_BLOCK
```

#### FB_DI.st
```iecst
FUNCTION_BLOCK FB_DI (* Univerzalni DI sa opcionim status signalom i fault dijagnostikom *) (*$GROUP=User,$CAT=User,$GROUPICON=User.png,$CATICON=User.png*)

(* -------------------------------------------------------------------------- *)
(* 1) Podrazumevane vrednosti po scan-u                                        *)
(* -------------------------------------------------------------------------- *)
DI_Output.Status := FALSE;
DI_Output.Alarm := FALSE;
DI_Output.Error := FALSE;
DI_Output.ManualActive := FALSE;
DI_Output.StatusSignalIn := DI_Input.StatusIn;

DI_Internal.FaultCondition := FALSE;
DI_Internal.AlarmCondition := FALSE;
DI_Internal.ResetAllowed := FALSE;

DI_Output.ResetAllowed := FALSE;
DI_Output.ConfigValid := TRUE;
DI_Output.ConfigFaultText := 'CONFIG_OK';
DI_Output.FaultCode := DI_Internal.FaultCode;
DI_Output.FaultText := DI_Internal.FaultText;
DI_Output.Diag := 'IDLE';

(* -------------------------------------------------------------------------- *)
(* 2) Validacija parametara i obrada sirovog signala                           *)
(* -------------------------------------------------------------------------- *)
DI_Internal.ConfigValid := TRUE;

IF DI_Param.DelayOn < T#0ms THEN
	DI_Internal.ConfigValid := FALSE;
	DI_Output.ConfigFaultText := 'DelayOn ne sme biti negativan';
END_IF;

IF DI_Param.DelayOff < T#0ms THEN
	DI_Internal.ConfigValid := FALSE;
	IF DI_Output.ConfigFaultText = 'CONFIG_OK' THEN
		DI_Output.ConfigFaultText := 'DelayOff ne sme biti negativan';
	END_IF;
END_IF;

IF DI_Param.InvertSignal THEN
	DI_Internal.SignalRaw := NOT DI_Input.SensorIn;
ELSE
	DI_Internal.SignalRaw := DI_Input.SensorIn;
END_IF;

(* -------------------------------------------------------------------------- *)
(* 3) Fault uslovi i reset politika (samo kada je Enable=TRUE)                 *)
(* -------------------------------------------------------------------------- *)
IF DI_Input.Enable THEN
	IF DI_Input.ManualAlarm THEN
		DI_Internal.FaultCondition := TRUE;
	END_IF;

	IF DI_Param.UseStatusInput AND (NOT DI_Input.StatusIn) THEN
		DI_Internal.FaultCondition := TRUE;
	END_IF;

	IF NOT DI_Internal.ConfigValid THEN
		DI_Internal.FaultCondition := TRUE;
	END_IF;

	DI_Internal.ResetAllowed := DI_Internal.FaultLatched AND (NOT DI_Internal.FaultCondition);

	IF DI_Input.ResetAlarm AND DI_Internal.ResetAllowed THEN
		DI_Internal.FaultLatched := FALSE;
		DI_Internal.FaultCode := DI_Constant.FLT_NONE;
	END_IF;

	IF DI_Internal.FaultCondition THEN
		IF NOT DI_Internal.FaultLatched THEN
			IF NOT DI_Internal.ConfigValid THEN
				DI_Internal.FaultCode := DI_Constant.FLT_CONFIG_INVALID;
			ELSIF DI_Input.ManualAlarm THEN
				DI_Internal.FaultCode := DI_Constant.FLT_MANUAL_ALARM;
			ELSE
				DI_Internal.FaultCode := DI_Constant.FLT_STATUS_INPUT;
			END_IF;
		END_IF;
		DI_Internal.FaultLatched := TRUE;
	END_IF;
ELSE
	DI_Internal.ResetAllowed := FALSE;
END_IF;

(* -------------------------------------------------------------------------- *)
(* 4) Glavna obrada po Enable/Manual/Auto granama                              *)
(* -------------------------------------------------------------------------- *)
IF NOT DI_Input.Enable THEN
	DI_Output.Value := FALSE;
	DI_Internal.SignalFiltered := FALSE;

	DI_Output.State := DI_Constant.ST_DISABLED;
	DI_Output.State_comment := 'Digitalni ulaz neaktivan';

	DI_Internal.TonOn(IN := FALSE, PT := DI_Param.DelayOn);
	DI_Internal.TonOff(IN := FALSE, PT := DI_Param.DelayOff);
ELSE
	IF DI_Input.EnableManual THEN
		DI_Output.Value := DI_Input.ManualValue;
		DI_Output.ManualActive := TRUE;

		DI_Internal.TonOn(IN := FALSE, PT := DI_Param.DelayOn);
		DI_Internal.TonOff(IN := FALSE, PT := DI_Param.DelayOff);
	ELSE
		DI_Output.ManualActive := FALSE;

		DI_Internal.TonOn(
			IN := DI_Internal.SignalRaw AND (NOT DI_Internal.SignalFiltered),
			PT := DI_Param.DelayOn
		);

		DI_Internal.TonOff(
			IN := (NOT DI_Internal.SignalRaw) AND DI_Internal.SignalFiltered,
			PT := DI_Param.DelayOff
		);

		IF (NOT DI_Internal.SignalFiltered) AND DI_Internal.SignalRaw THEN
			IF (DI_Param.DelayOn = T#0s) OR DI_Internal.TonOn.Q THEN
				DI_Internal.SignalFiltered := TRUE;
			END_IF;
		END_IF;

		IF DI_Internal.SignalFiltered AND (NOT DI_Internal.SignalRaw) THEN
			IF (DI_Param.DelayOff = T#0s) OR DI_Internal.TonOff.Q THEN
				DI_Internal.SignalFiltered := FALSE;
			END_IF;
		END_IF;

		DI_Output.Value := DI_Internal.SignalFiltered;
	END_IF;

	DI_Internal.AlarmCondition := FALSE;

	IF DI_Output.Value AND DI_Param.AlarmOnTrue THEN
		DI_Internal.AlarmCondition := TRUE;
	END_IF;

	IF (NOT DI_Output.Value) AND DI_Param.AlarmOnFalse THEN
		DI_Internal.AlarmCondition := TRUE;
	END_IF;

	IF DI_Internal.FaultLatched THEN
		DI_Output.Status := FALSE;
		DI_Output.Alarm := DI_Internal.AlarmCondition;
		DI_Output.Error := TRUE;

		IF DI_Input.EnableManual THEN
			DI_Output.State := DI_Constant.ST_MAN_FAULT;
		ELSE
			DI_Output.State := DI_Constant.ST_AUTO_FAULT;
		END_IF;
		DI_Output.State_comment := DI_Param.TextFault;
	ELSE
		DI_Output.Status := TRUE;
		DI_Output.Alarm := DI_Internal.AlarmCondition;
		DI_Output.Error := FALSE;

		IF DI_Input.EnableManual THEN
			IF DI_Internal.AlarmCondition THEN
				DI_Output.State := DI_Constant.ST_MAN_ALARM;
				DI_Output.State_comment := DI_Param.TextAlarm;
			ELSE
				IF DI_Output.Value THEN
					DI_Output.State := DI_Constant.ST_MAN_TRUE;
					DI_Output.State_comment := DI_Param.TextTrue;
				ELSE
					DI_Output.State := DI_Constant.ST_MAN_FALSE;
					DI_Output.State_comment := DI_Param.TextFalse;
				END_IF;
			END_IF;
		ELSE
			IF DI_Internal.AlarmCondition THEN
				DI_Output.State := DI_Constant.ST_AUTO_ALARM;
				DI_Output.State_comment := DI_Param.TextAlarm;
			ELSE
				IF DI_Output.Value THEN
					DI_Output.State := DI_Constant.ST_AUTO_TRUE;
					DI_Output.State_comment := DI_Param.TextTrue;
				ELSE
					DI_Output.State := DI_Constant.ST_AUTO_FALSE;
					DI_Output.State_comment := DI_Param.TextFalse;
				END_IF;
			END_IF;
		END_IF;
	END_IF;
END_IF;

(* -------------------------------------------------------------------------- *)
(* 5) Fault tekst i dijagnostika                                               *)
(* -------------------------------------------------------------------------- *)
CASE DI_Internal.FaultCode OF
	0:
		DI_Internal.FaultText := 'FLT_NONE - nema memorisanog fault-a';
	1:
		DI_Internal.FaultText := 'FLT_MANUAL_ALARM - aktivan ManualAlarm ulaz';
	2:
		DI_Internal.FaultText := 'FLT_STATUS_INPUT - StatusIn je FALSE uz aktivan UseStatusInput';
	3:
		DI_Internal.FaultText := 'FLT_CONFIG_INVALID - nevalidni Delay parametri';
ELSE
	DI_Internal.FaultText := 'FLT_UNKNOWN - nepoznat fault kod';
END_CASE;

IF NOT DI_Input.Enable THEN
	DI_Internal.Diag := 'DISABLED';
ELSIF NOT DI_Internal.ConfigValid THEN
	DI_Internal.Diag := 'CONFIG_INVALID';
ELSIF DI_Internal.FaultLatched THEN
	DI_Internal.Diag := 'FAULT_LATCHED';
ELSIF DI_Input.EnableManual THEN
	IF DI_Internal.AlarmCondition THEN
		DI_Internal.Diag := 'MANUAL_ALARM';
	ELSE
		DI_Internal.Diag := 'MANUAL_OK';
	END_IF;
ELSE
	IF DI_Internal.AlarmCondition THEN
		DI_Internal.Diag := 'AUTO_ALARM';
	ELSE
		DI_Internal.Diag := 'AUTO_OK';
	END_IF;
END_IF;

(* -------------------------------------------------------------------------- *)
(* 6) Zavrsno mapiranje dijagnostickih izlaza                                  *)
(* -------------------------------------------------------------------------- *)
DI_Output.FaultLatched := DI_Internal.FaultLatched;
DI_Output.FaultCondition := DI_Internal.FaultCondition;
DI_Output.AlarmCondition := DI_Internal.AlarmCondition;
DI_Output.ResetAllowed := DI_Internal.ResetAllowed;
DI_Output.ConfigValid := DI_Internal.ConfigValid;
DI_Output.FaultCode := DI_Internal.FaultCode;
DI_Output.FaultText := DI_Internal.FaultText;
DI_Output.Diag := DI_Internal.Diag;

END_FUNCTION_BLOCK
```
